REGION Network 2: MOVIMIENTO DE DATOS
   RUNG wire#powerrail
      Move(in := "FLUJO_FB_DB".SEÑAL_INGENIERIA, out1 => "flujo")
   END_RUNG
   RUNG wire#powerrail
      Move(in := "PRESION_LIQUIDO_FB_DB".SEÑAL_INGENIERIA, out1 => "presion")
   END_RUNG
   RUNG wire#powerrail
      Move(in := "valvula", out1 => "Consigna apertura Valvula Proporcional")
   END_RUNG
   RUNG wire#powerrail
      Move(in := "TEMPERATURA_FB_DB".SEÑAL_INGENIERIA, out1 => "temperatura")
   END_RUNG
   RUNG wire#powerrail
      Move(in := "PESO_FB_DB".SEÑAL_INGENIERIA, out1 => "peso tanque")
   END_RUNG
   RUNG wire#powerrail
      Move(in := "NIVEL_FB_DB".SEÑAL_INGENIERIA, out1 => "nivel_tanque")
   END_RUNG
   RUNG wire#powerrail
      Move(in := "bomba", out1 => "Consigna Velocidad Variador")
   END_RUNG
   // the same network as SCL:
   "flujo" := "FLUJO_FB_DB".SEÑAL_INGENIERIA;
   "presion" := "PRESION_LIQUIDO_FB_DB".SEÑAL_INGENIERIA;
   "Consigna apertura Valvula Proporcional" := "valvula";
   "temperatura" := "TEMPERATURA_FB_DB".SEÑAL_INGENIERIA;
   "peso tanque" := "PESO_FB_DB".SEÑAL_INGENIERIA;
   "nivel_tanque" := "NIVEL_FB_DB".SEÑAL_INGENIERIA;
   "Consigna Velocidad Variador" := "bomba";
END_REGION

REGION Network 3: PID NIVEL
   RUNG wire#powerrail
      Contact( "Tag_12" )
      "Smith_please_DB_1"(Sensor := "nivel_cal", Ref := "ref_lgr_nivel", Bomba => "bomba")
   END_RUNG
   // the same network as SCL:
   IF "Tag_12" THEN
       "Smith_please_DB_1"(Sensor := "nivel_cal", Ref := "ref_lgr_nivel", Bomba => "bomba");   // "Smith_please"
   END_IF;
END_REGION

REGION Network 4: ALARMAS
   RUNG wire#powerrail
      "ALARMAS"()
   END_RUNG
   // the same network as SCL:
   "ALARMAS"();
END_REGION

REGION Network 5: CARACTERIZACION Y CALIBRACION
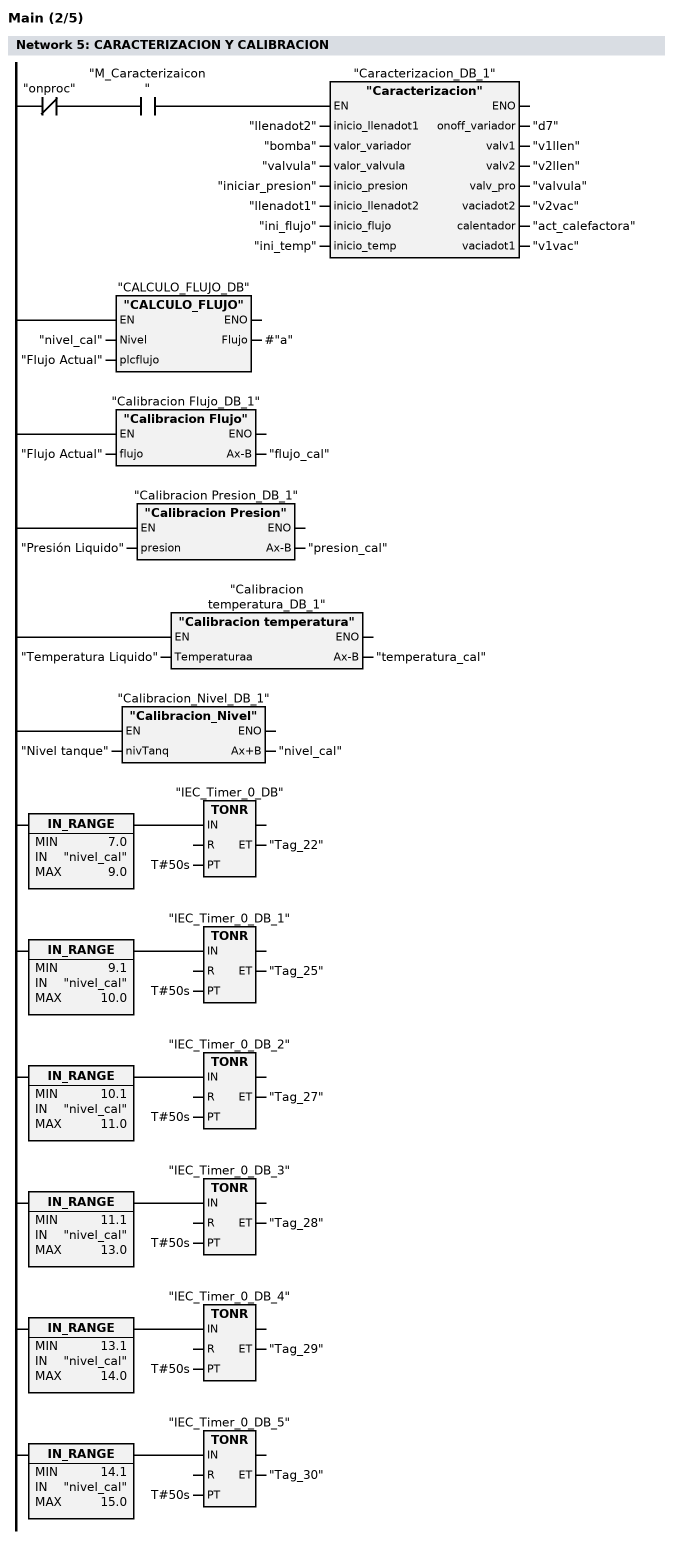
   IF NOT "onproc" AND "M_Caracterizaicon" THEN
       "Caracterizacion_DB_1"(inicio_llenadot1 := "llenadot2",   // "Caracterizacion"
                              valor_variador := "bomba",
                              valor_valvula := "valvula",
                              inicio_presion := "iniciar_presion",
                              inicio_llenadot2 := "llenadot1",
                              inicio_flujo := "ini_flujo",
                              inicio_temp := "ini_temp",
                              onoff_variador => "d7",
                              valv1 => "v1llen",
                              valv2 => "v2llen",
                              valv_pro => "valvula",
                              vaciadot2 => "v2vac",
                              calentador => "act_calefactora",
                              vaciadot1 => "v1vac");
   END_IF;
   "CALCULO_FLUJO_DB"(Nivel := "nivel_cal", plcflujo := "Flujo Actual", Flujo => #"a");   // "CALCULO_FLUJO"
   "Calibracion Flujo_DB_1"(flujo := "Flujo Actual", "Ax-B" => "flujo_cal");   // "Calibracion Flujo"
   "Calibracion Presion_DB_1"(presion := "Presión Liquido", "Ax-B" => "presion_cal");   // "Calibracion Presion"
   "Calibracion temperatura_DB_1"(Temperaturaa := "Temperatura Liquido", "Ax-B" => "temperatura_cal");   // "Calibracion temperatura"
   "Calibracion_Nivel_DB_1"(nivTanq := "Nivel tanque", "Ax+B" => "nivel_cal");   // "Calibracion_Nivel"
   "IEC_Timer_0_DB".TONR(IN := (7.0 <= "nivel_cal") AND ("nivel_cal" <= 9.0), PT := T#50s, ET => "Tag_22");
   "IEC_Timer_0_DB_1".TONR(IN := (9.1 <= "nivel_cal") AND ("nivel_cal" <= 10.0), PT := T#50s, ET => "Tag_25");
   "IEC_Timer_0_DB_2".TONR(IN := (10.1 <= "nivel_cal") AND ("nivel_cal" <= 11.0), PT := T#50s, ET => "Tag_27");
   "IEC_Timer_0_DB_3".TONR(IN := (11.1 <= "nivel_cal") AND ("nivel_cal" <= 13.0), PT := T#50s, ET => "Tag_28");
   "IEC_Timer_0_DB_4".TONR(IN := (13.1 <= "nivel_cal") AND ("nivel_cal" <= 14.0), PT := T#50s, ET => "Tag_29");
   "IEC_Timer_0_DB_5".TONR(IN := (14.1 <= "nivel_cal") AND ("nivel_cal" <= 15.0), PT := T#50s, ET => "Tag_30");
END_REGION

REGION Network 6: ON OFF PESO
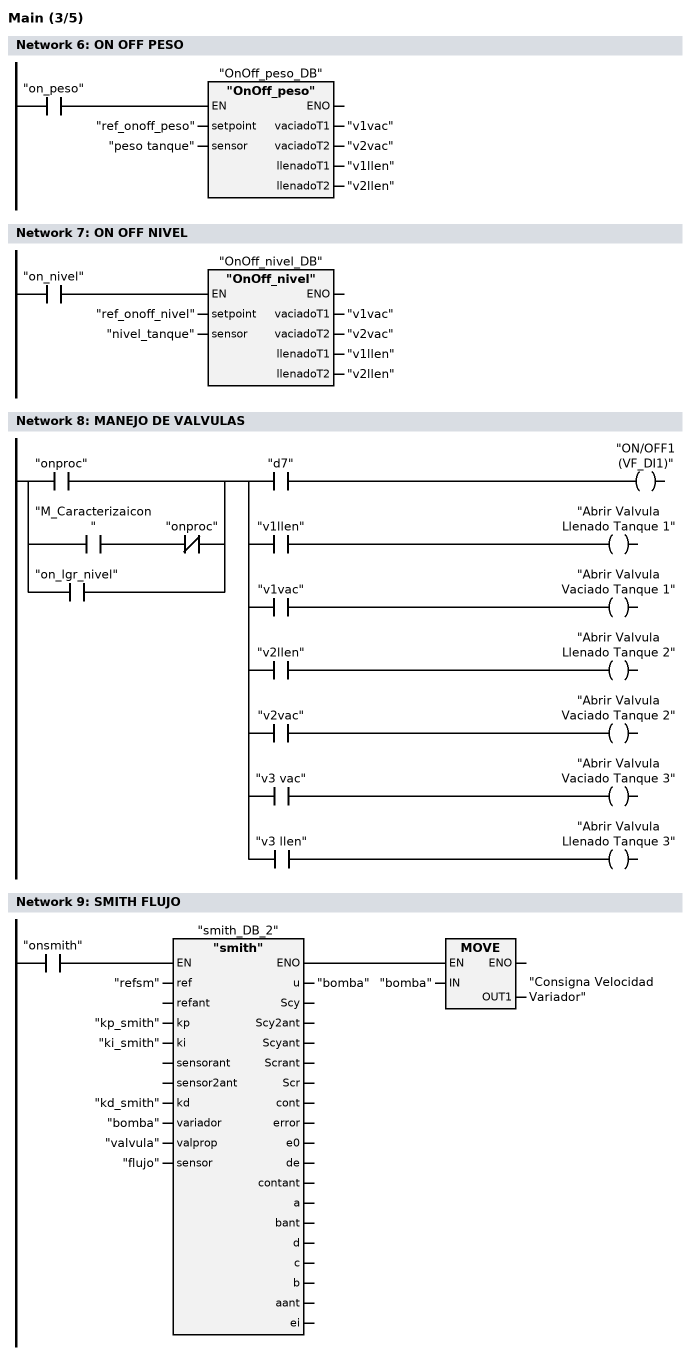
   RUNG wire#powerrail
      Contact( "on_peso" )
      "OnOff_peso_DB"(setpoint := "ref_onoff_peso", sensor := "peso tanque", vaciadoT1 => "v1vac", vaciadoT2 => "v2vac", llenadoT1 => "v1llen", llenadoT2 => "v2llen")
   END_RUNG
   // the same network as SCL:
   IF "on_peso" THEN
       "OnOff_peso_DB"(setpoint := "ref_onoff_peso",   // "OnOff_peso"
                       sensor := "peso tanque",
                       vaciadoT1 => "v1vac",
                       vaciadoT2 => "v2vac",
                       llenadoT1 => "v1llen",
                       llenadoT2 => "v2llen");
   END_IF;
END_REGION

REGION Network 7: ON OFF NIVEL
   RUNG wire#powerrail
      Contact( "on_nivel" )
      "OnOff_nivel_DB"(setpoint := "ref_onoff_nivel", sensor := "nivel_tanque", vaciadoT1 => "v1vac", vaciadoT2 => "v2vac", llenadoT1 => "v1llen", llenadoT2 => "v2llen")
   END_RUNG
   // the same network as SCL:
   IF "on_nivel" THEN
       "OnOff_nivel_DB"(setpoint := "ref_onoff_nivel",   // "OnOff_nivel"
                        sensor := "nivel_tanque",
                        vaciadoT1 => "v1vac",
                        vaciadoT2 => "v2vac",
                        llenadoT1 => "v1llen",
                        llenadoT2 => "v2llen");
   END_IF;
END_REGION

REGION Network 8: MANEJO DE VALVULAS
   RUNG wire#powerrail
      Contact( "onproc" )
      wire#w1
      Contact( "d7" )
      Coil( "ON/OFF1 (VF_DI1)" )
   END_RUNG
   RUNG wire#powerrail
      Contact( "M_Caracterizaicon" )
      I_Contact( "onproc" )
   END_RUNG wire#w1
   RUNG wire#powerrail
      Contact( "on_lgr_nivel" )
   END_RUNG wire#w1
   RUNG wire#w1
      Contact( "v1llen" )
      Coil( "Abrir Valvula Llenado Tanque 1" )
   END_RUNG
   RUNG wire#w1
      Contact( "v1vac" )
      Coil( "Abrir Valvula Vaciado Tanque 1" )
   END_RUNG
   RUNG wire#w1
      Contact( "v2llen" )
      Coil( "Abrir Valvula Llenado Tanque 2" )
   END_RUNG
   RUNG wire#w1
      Contact( "v2vac" )
      Coil( "Abrir Valvula Vaciado Tanque 2" )
   END_RUNG
   RUNG wire#w1
      Contact( "v3 vac" )
      Coil( "Abrir Valvula Vaciado Tanque 3" )
   END_RUNG
   RUNG wire#w1
      Contact( "v3 llen" )
      Coil( "Abrir Valvula Llenado Tanque 3" )
   END_RUNG
   // the same network as SCL:
   #_w1 := "onproc" OR ("M_Caracterizaicon" AND NOT "onproc") OR "on_lgr_nivel";
   "ON/OFF1 (VF_DI1)" := #_w1 AND "d7";
   "Abrir Valvula Llenado Tanque 1" := #_w1 AND "v1llen";
   "Abrir Valvula Vaciado Tanque 1" := #_w1 AND "v1vac";
   "Abrir Valvula Llenado Tanque 2" := #_w1 AND "v2llen";
   "Abrir Valvula Vaciado Tanque 2" := #_w1 AND "v2vac";
   "Abrir Valvula Vaciado Tanque 3" := #_w1 AND "v3 vac";
   "Abrir Valvula Llenado Tanque 3" := #_w1 AND "v3 llen";
END_REGION

REGION Network 9: SMITH FLUJO
   RUNG wire#powerrail
      Contact( "onsmith" )
      "smith_DB_2"(ref := "refsm", refant :=, kp := "kp_smith", ki := "ki_smith", sensorant :=, sensor2ant :=, kd := "kd_smith", variador := "bomba", valprop := "valvula", sensor := "flujo", u => "bomba", Scy =>, Scy2ant =>, Scyant =>, Scrant =>, Scr =>, cont =>, error =>, e0 =>, de =>, contant =>, "a" =>, bant =>, d =>, c =>, "b" =>, aant =>, ei =>)
      Move(in := "bomba", out1 => "Consigna Velocidad Variador")
   END_RUNG
   // the same network as SCL:
   "smith_DB_2"(EN := "onsmith",   // "smith"
                ref := "refsm",
                kp := "kp_smith",
                ki := "ki_smith",
                kd := "kd_smith",
                variador := "bomba",
                valprop := "valvula",
                sensor := "flujo",
                u => "bomba",
                ENO => #_w1);
   IF #_w1 THEN "Consigna Velocidad Variador" := "bomba"; END_IF;
END_REGION

REGION Network 10: ON OFF TEMPERATURA
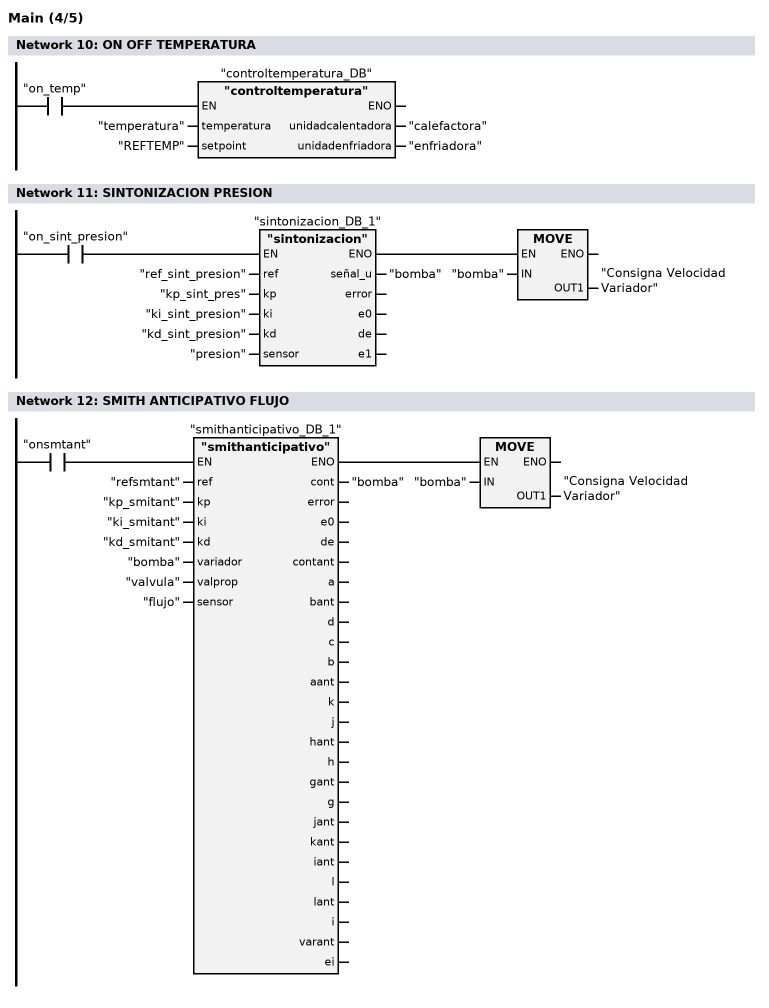
   RUNG wire#powerrail
      Contact( "on_temp" )
      "controltemperatura_DB"(temperatura := "temperatura", setpoint := "REFTEMP", unidadcalentadora => "calefactora", unidadenfriadora => "enfriadora")
   END_RUNG
   // the same network as SCL:
   IF "on_temp" THEN
       "controltemperatura_DB"(temperatura := "temperatura",   // "controltemperatura"
                               setpoint := "REFTEMP",
                               unidadcalentadora => "calefactora",
                               unidadenfriadora => "enfriadora");
   END_IF;
END_REGION

REGION Network 11: SINTONIZACION PRESION
   RUNG wire#powerrail
      Contact( "on_sint_presion" )
      "sintonizacion_DB_1"(ref := "ref_sint_presion", kp := "kp_sint_pres", ki := "ki_sint_presion", kd := "kd_sint_presion", sensor := "presion", señal_u => "bomba", error =>, e0 =>, de =>, e1 =>)
      Move(in := "bomba", out1 => "Consigna Velocidad Variador")
   END_RUNG
   // the same network as SCL:
   "sintonizacion_DB_1"(EN := "on_sint_presion",   // "sintonizacion"
                        ref := "ref_sint_presion",
                        kp := "kp_sint_pres",
                        ki := "ki_sint_presion",
                        kd := "kd_sint_presion",
                        sensor := "presion",
                        señal_u => "bomba",
                        ENO => #_w1);
   IF #_w1 THEN "Consigna Velocidad Variador" := "bomba"; END_IF;
END_REGION

REGION Network 12: SMITH ANTICIPATIVO FLUJO
   RUNG wire#powerrail
      Contact( "onsmtant" )
      "smithanticipativo_DB_1"(ref := "refsmtant", kp := "kp_smitant", ki := "ki_smitant", kd := "kd_smitant", variador := "bomba", valprop := "valvula", sensor := "flujo", cont => "bomba", error =>, e0 =>, de =>, contant =>, "a" =>, bant =>, d =>, c =>, "b" =>, aant =>, k =>, j =>, hant =>, h =>, gant =>, g =>, jant =>, kant =>, iant =>, l =>, lant =>, i =>, varant =>, ei =>)
      Move(in := "bomba", out1 => "Consigna Velocidad Variador")
   END_RUNG
   // the same network as SCL:
   "smithanticipativo_DB_1"(EN := "onsmtant",   // "smithanticipativo"
                           ref := "refsmtant",
                           kp := "kp_smitant",
                           ki := "ki_smitant",
                           kd := "kd_smitant",
                           variador := "bomba",
                           valprop := "valvula",
                           sensor := "flujo",
                           cont => "bomba",
                           ENO => #_w1);
   IF #_w1 THEN "Consigna Velocidad Variador" := "bomba"; END_IF;
END_REGION

REGION Network 13: FUZZY PRESION
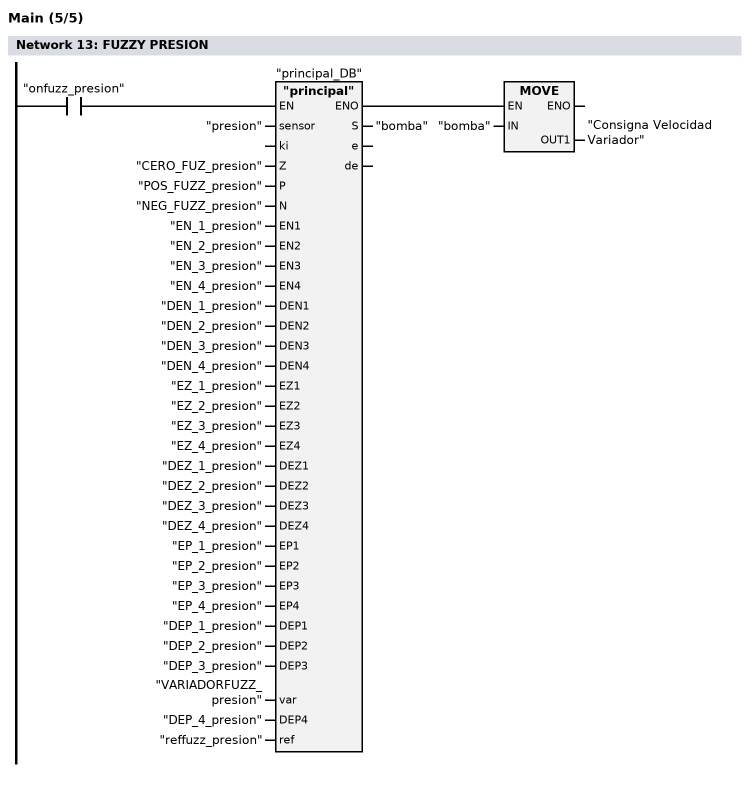
   RUNG wire#powerrail
      Contact( "onfuzz_presion" )
      "principal_DB"(sensor := "presion", ki :=, Z := "CERO_FUZ_presion", P := "POS_FUZZ_presion", N := "NEG_FUZZ_presion", EN1 := "EN_1_presion", EN2 := "EN_2_presion", EN3 := "EN_3_presion", EN4 := "EN_4_presion", DEN1 := "DEN_1_presion", DEN2 := "DEN_2_presion", DEN3 := "DEN_3_presion", DEN4 := "DEN_4_presion", EZ1 := "EZ_1_presion", EZ2 := "EZ_2_presion", EZ3 := "EZ_3_presion", EZ4 := "EZ_4_presion", DEZ1 := "DEZ_1_presion", DEZ2 := "DEZ_2_presion", DEZ3 := "DEZ_3_presion", DEZ4 := "DEZ_4_presion", EP1 := "EP_1_presion", EP2 := "EP_2_presion", EP3 := "EP_3_presion", EP4 := "EP_4_presion", DEP1 := "DEP_1_presion", DEP2 := "DEP_2_presion", DEP3 := "DEP_3_presion", var := "VARIADORFUZZ_presion", DEP4 := "DEP_4_presion", ref := "reffuzz_presion", S => "bomba", "e" =>, de =>)
      Move(in := "bomba", out1 => "Consigna Velocidad Variador")
   END_RUNG
   // the same network as SCL:
   "principal_DB"(EN := "onfuzz_presion",   // "principal"
                  sensor := "presion",
                  Z := "CERO_FUZ_presion",
                  P := "POS_FUZZ_presion",
                  N := "NEG_FUZZ_presion",
                  EN1 := "EN_1_presion",
                  EN2 := "EN_2_presion",
                  EN3 := "EN_3_presion",
                  EN4 := "EN_4_presion",
                  DEN1 := "DEN_1_presion",
                  DEN2 := "DEN_2_presion",
                  DEN3 := "DEN_3_presion",
                  DEN4 := "DEN_4_presion",
                  EZ1 := "EZ_1_presion",
                  EZ2 := "EZ_2_presion",
                  EZ3 := "EZ_3_presion",
                  EZ4 := "EZ_4_presion",
                  DEZ1 := "DEZ_1_presion",
                  DEZ2 := "DEZ_2_presion",
                  DEZ3 := "DEZ_3_presion",
                  DEZ4 := "DEZ_4_presion",
                  EP1 := "EP_1_presion",
                  EP2 := "EP_2_presion",
                  EP3 := "EP_3_presion",
                  EP4 := "EP_4_presion",
                  DEP1 := "DEP_1_presion",
                  DEP2 := "DEP_2_presion",
                  DEP3 := "DEP_3_presion",
                  var := "VARIADORFUZZ_presion",
                  DEP4 := "DEP_4_presion",
                  ref := "reffuzz_presion",
                  S => "bomba",
                  ENO => #_w1);
   IF #_w1 THEN "Consigna Velocidad Variador" := "bomba"; END_IF;
END_REGION
END_ORGANIZATION_BLOCK

ORGANIZATION_BLOCK "Cyclic interrupt"   // OB30, LAD, CyclicInterrupt
{ S7_Optimized_Access := 'TRUE' }
VERSION : 0.1
   VAR_INPUT
      Initial_Call : Bool;   // Initial call of this OB
      Event_Count : Int;   // Events discarded
   END_VAR
   VAR_TEMP
      PIDDT : Bool;
   END_VAR
BEGIN

REGION Network 2
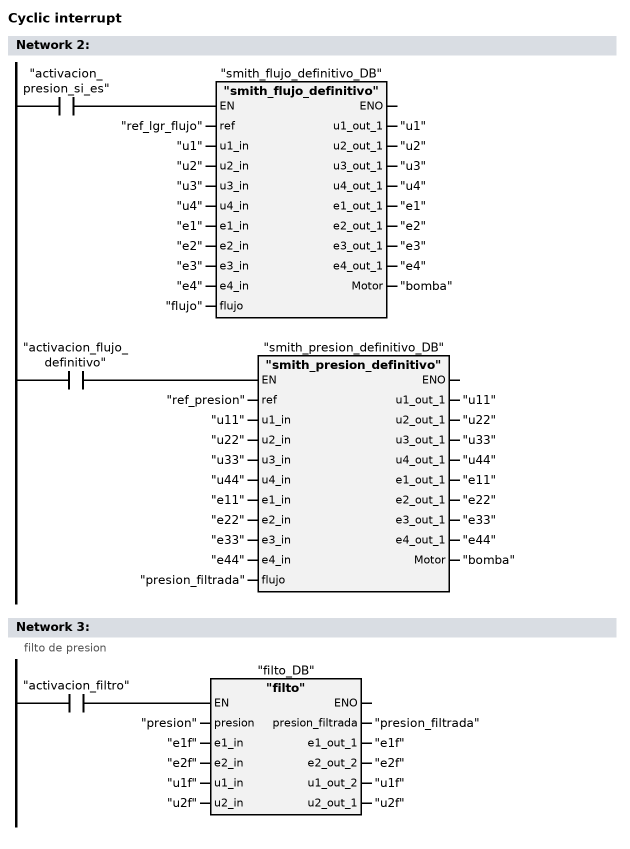
   RUNG wire#powerrail
      Contact( "activacion_presion_si_es" )
      "smith_flujo_definitivo_DB"(ref := "ref_lgr_flujo", u1_in := "u1", u2_in := "u2", u3_in := "u3", u4_in := "u4", e1_in := "e1", e2_in := "e2", e3_in := "e3", e4_in := "e4", flujo := "flujo", u1_out_1 => "u1", u2_out_1 => "u2", u3_out_1 => "u3", u4_out_1 => "u4", e1_out_1 => "e1", e2_out_1 => "e2", e3_out_1 => "e3", e4_out_1 => "e4", Motor => "bomba")
   END_RUNG
   RUNG wire#powerrail
      Contact( "activacion_flujo_definitivo" )
      "smith_presion_definitivo_DB"(ref := "ref_presion", u1_in := "u11", u2_in := "u22", u3_in := "u33", u4_in := "u44", e1_in := "e11", e2_in := "e22", e3_in := "e33", e4_in := "e44", flujo := "presion_filtrada", u1_out_1 => "u11", u2_out_1 => "u22", u3_out_1 => "u33", u4_out_1 => "u44", e1_out_1 => "e11", e2_out_1 => "e22", e3_out_1 => "e33", e4_out_1 => "e44", Motor => "bomba")
   END_RUNG
   // the same network as SCL:
   IF "activacion_presion_si_es" THEN
       "smith_flujo_definitivo_DB"(ref := "ref_lgr_flujo",   // "smith_flujo_definitivo"
                               u1_in := "u1",
                               u2_in := "u2",
                               u3_in := "u3",
                               u4_in := "u4",
                               e1_in := "e1",
                               e2_in := "e2",
                               e3_in := "e3",
                               e4_in := "e4",
                               flujo := "flujo",
                               u1_out_1 => "u1",
                               u2_out_1 => "u2",
                               u3_out_1 => "u3",
                               u4_out_1 => "u4",
                               e1_out_1 => "e1",
                               e2_out_1 => "e2",
                               e3_out_1 => "e3",
                               e4_out_1 => "e4",
                               Motor => "bomba");
   END_IF;
   IF "activacion_flujo_definitivo" THEN
       "smith_presion_definitivo_DB"(ref := "ref_presion",   // "smith_presion_definitivo"
                               u1_in := "u11",
                               u2_in := "u22",
                               u3_in := "u33",
                               u4_in := "u44",
                               e1_in := "e11",
                               e2_in := "e22",
                               e3_in := "e33",
                               e4_in := "e44",
                               flujo := "presion_filtrada",
                               u1_out_1 => "u11",
                               u2_out_1 => "u22",
                               u3_out_1 => "u33",
                               u4_out_1 => "u44",
                               e1_out_1 => "e11",
                               e2_out_1 => "e22",
                               e3_out_1 => "e33",
                               e4_out_1 => "e44",
                               Motor => "bomba");
   END_IF;
END_REGION

REGION Network 3
   // filto de presion
   RUNG wire#powerrail
      Contact( "activacion_filtro" )
      "filto_DB"(presion := "presion", e1_in := "e1f", e2_in := "e2f", u1_in := "u1f", u2_in := "u2f", presion_filtrada => "presion_filtrada", e1_out_1 => "e1f", e2_out_2 => "e2f", u1_out_2 => "u1f", u2_out_1 => "u2f")
   END_RUNG
   // the same network as SCL:
   IF "activacion_filtro" THEN
       "filto_DB"(presion := "presion",   // "filto"
                  e1_in := "e1f",
                  e2_in := "e2f",
                  u1_in := "u1f",
                  u2_in := "u2f",
                  presion_filtrada => "presion_filtrada",
                  e1_out_1 => "e1f",
                  e2_out_2 => "e2f",
                  u1_out_2 => "u1f",
                  u2_out_1 => "u2f");
   END_IF;
END_REGION
END_ORGANIZATION_BLOCK

ORGANIZATION_BLOCK "Startup"   // OB100, LAD, Startup
TITLE = "Complete Restart"
{ S7_Optimized_Access := 'TRUE' }
VERSION : 0.1
   VAR_INPUT
      LostRetentive : Bool;   // True if retentive data are lost
      LostRTC : Bool;   // True if date and time are lost
   END_VAR
BEGIN

REGION Network 1
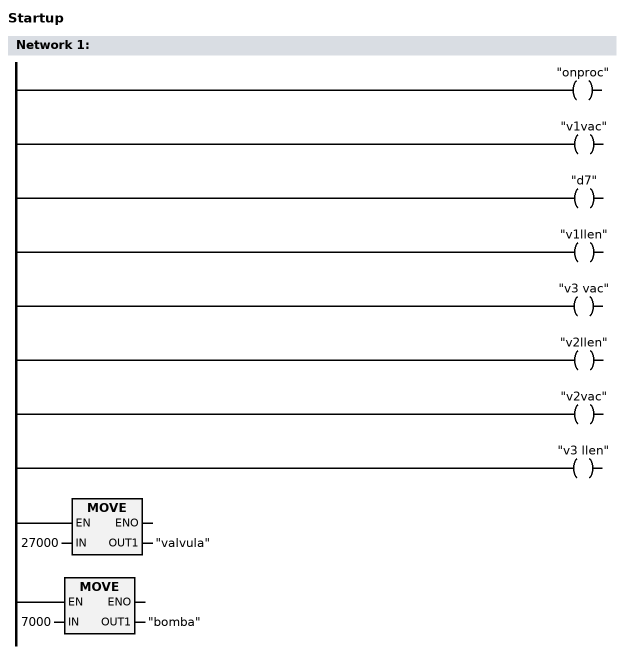
   RUNG wire#powerrail
      Coil( "onproc" )
   END_RUNG
   RUNG wire#powerrail
      Coil( "v1vac" )
   END_RUNG
   RUNG wire#powerrail
      Coil( "d7" )
   END_RUNG
   RUNG wire#powerrail
      Coil( "v1llen" )
   END_RUNG
   RUNG wire#powerrail
      Coil( "v3 vac" )
   END_RUNG
   RUNG wire#powerrail
      Coil( "v2llen" )
   END_RUNG
   RUNG wire#powerrail
      Coil( "v2vac" )
   END_RUNG
   RUNG wire#powerrail
      Coil( "v3 llen" )
   END_RUNG
   RUNG wire#powerrail
      Move(in := 27000, out1 => "valvula")
   END_RUNG
   RUNG wire#powerrail
      Move(in := 7000, out1 => "bomba")
   END_RUNG
   // the same network as SCL:
   "onproc" := TRUE;
   "v1vac" := TRUE;
   "d7" := TRUE;
   "v1llen" := TRUE;
   "v3 vac" := TRUE;
   "v2llen" := TRUE;
   "v2vac" := TRUE;
   "v3 llen" := TRUE;
   "valvula" := 27000;
   "bomba" := 7000;
END_REGION
END_ORGANIZATION_BLOCK

(* ===== HMI "HMI_RT_1" =====
system functions are stored by id; their names below are inferred from use
connection "HMI_Conexión_2": ETHERNET, S7_1500_OMS

HMI tags "Tabla de variables estándar"
   "Número_imagen_variable" : UInt, internal
   "v1llen" : Bool = PLC v1llen AT %M2.3, 1 s
   "v1vac" : Bool = PLC v1vac AT %M2.4, 1 s
   "v2llen" : Bool = PLC v2llen AT %M2.5, 1 s
   "v2vac" : Bool = PLC v2vac AT %M2.6, 1 s
   "v3" : Bool = PLC "v3 vac" AT %M5.0, 1 s
   "valvula" : Int = PLC valvula AT %MW8, 1 s
   "onproc" : Bool = PLC onproc AT %M2.7, 1 s
   "d7" : Bool = PLC d7 AT %M3.0, 1 s
   "bomba" : Int = PLC bomba AT %MW6, 1 s
   "onsint" : Bool = PLC onsint AT %M5.3, 1 s
   "onfuzz" : Bool = PLC onfuzz AT %M5.1, 1 s
   "Nivel tanque" : Int = PLC "Nivel tanque" AT %IW112, 1 s
   "velmotor" : Word = PLC velmotor AT %MW26, 1 s
   "presion" : Real = PLC presion AT %MD10, 1 s
   "flujo" : Real = PLC flujo AT %MD14, 1 s
   "refsint" : Real = PLC refsint AT %MD24, 1 s
   "reflgr" : Real = PLC reflgr AT %MD26, 1 s
   "onlgr" : Bool = PLC onlgr AT %M5.6, 1 s
   "onsmith" : Bool = PLC onsmith AT %M5.4, 1 s
   "onsmtant" : Bool = PLC onsmtant AT %M5.5, 1 s
   "refsmtant" : Real = PLC refsmtant AT %MD28, 1 s
   "reffuzz" : Real = PLC reffuzz AT %MD22, 1 s
   "temperatura" : Real = PLC temperatura AT %MD16, 1 s
   "REFTEMP" : Real = PLC REFTEMP AT %MD30, 1 s
   "on_temp" : Bool = PLC on_temp AT %M5.7, 1 s
   "Activar Unidad Enfriadora" : Bool = PLC "Activar Unidad Enfriadora" AT %Q1.7, 1 s
   "Activar Unidad Calefactora" : Bool = PLC "Activar Unidad Calefactora" AT %Q1.6, 1 s
   "Abrir Valvula Vaciado Tanque 3" : Bool = PLC "Abrir Valvula Vaciado Tanque 3" AT %Q1.5, 1 s
   "Abrir Valvula Llenado Tanque 3" : Bool = PLC "Abrir Valvula Llenado Tanque 3" AT %Q1.4, 1 s
   "Temperatura Liquido" : Int = PLC "Temperatura Liquido" AT %IW106, 1 s
   "kp_sint" : Real = PLC kp_sint AT %MD34, 1 s
   "ki_sint" : Real = PLC ki_sint AT %MD38, 1 s
   "kd_sint" : Real = PLC kd_sint AT %MD42, 1 s
   "Consigna apertura Valvula Proporcional" : Int = PLC "Consigna apertura Valvula Proporcional" AT %QW106, 1 s
   "Consigna Velocidad Variador" : Int = PLC "Consigna Velocidad Variador" AT %QW104, 1 s
   "Switch de Nivel Alto Tanque 1 (NC)" : Bool = PLC "Switch de Nivel Alto Tanque 1 (NC)" AT %I1.3, 1 s
   "Switch de Nivel Bajo Tanque 1 (NO)" : Bool = PLC "Switch de Nivel Bajo Tanque 1 (NO)" AT %I1.2, 1 s
   "Abrir Valvula Llenado Tanque 1" : Bool = PLC "Abrir Valvula Llenado Tanque 1" AT %Q1.0, 1 s
   "Abrir Valvula Llenado Tanque 2" : Bool = PLC "Abrir Valvula Llenado Tanque 2" AT %Q1.2, 1 s
   "Abrir Valvula Vaciado Tanque 1" : Bool = PLC "Abrir Valvula Vaciado Tanque 1" AT %Q1.1, 1 s
   "Abrir Valvula Vaciado Tanque 2" : Bool = PLC "Abrir Valvula Vaciado Tanque 2" AT %Q1.3, 1 s
   "kp_lgr" : Real = PLC kp_lgr AT %MD46, 1 s
   "ki_lgr" : Real = PLC ki_lgr AT %MD54, 1 s
   "kd_lgr" : Real = PLC kd_lgr AT %MD58, 1 s
   "refsm" : Real = PLC refsm AT %MD20, 1 s
   "kp_smith" : Real = PLC kp_smith AT %MD62, 1 s
   "ki_smith" : Real = PLC ki_smith AT %MD66, 1 s
   "kd_smith" : Real = PLC kd_smith AT %MD70, 1 s
   "kp_smitant" : Real = PLC kp_smitant AT %MD74, 1 s
   "ki_smitant" : Real = PLC ki_smitant AT %MD78, 1 s
   "kd_smitant" : Real = PLC kd_smitant AT %MD82, 1 s
   "EN_1" : Real = PLC EN_1 AT %MD98, 1 s
   "EN_2" : Real = PLC EN_2 AT %MD102, 1 s
   "EN_3" : Real = PLC EN_3 AT %MD106, 1 s
   "EN_4" : Real = PLC EN_4 AT %MD110, 1 s
   "EZ_1" : Real = PLC EZ_1 AT %MD130, 1 s
   "EZ_2" : Real = PLC EZ_2 AT %MD134, 1 s
   "EZ_3" : Real = PLC EZ_3 AT %MD138, 1 s
   "EZ_4" : Real = PLC EZ_4 AT %MD142, 1 s
   "EP_1" : Real = PLC EP_1 AT %MD162, 1 s
   "EP_2" : Real = PLC EP_2 AT %MD166, 1 s
   "EP_3" : Real = PLC EP_3 AT %MD170, 1 s
   "EP_4" : Real = PLC EP_4 AT %MD174, 1 s
   "DEN_1" : Real = PLC DEN_1 AT %MD114, 1 s
   "DEN_2" : Real = PLC DEN_2 AT %MD118, 1 s
   "DEN_3" : Real = PLC DEN_3 AT %MD122, 1 s
   "DEN_4" : Real = PLC DEN_4 AT %MD126, 1 s
   "DEZ_1" : Real = PLC DEZ_1 AT %MD146, 1 s
   "DEZ_2" : Real = PLC DEZ_2 AT %MD150, 1 s
   "DEZ_3" : Real = PLC DEZ_3 AT %MD154, 1 s
   "DEZ_4" : Real = PLC DEZ_4 AT %MD158, 1 s
   "DEP_1" : Real = PLC DEP_1 AT %MD178, 1 s
   "DEP_2" : Real = PLC DEP_2 AT %MD182, 1 s
   "DEP_3" : Real = PLC DEP_3 AT %MD186, 1 s
   "DEP_4" : Real = PLC DEP_4 AT %MD194, 1 s
   "NEG_FUZZ" : Real = PLC NEG_FUZZ AT %MD94, 1 s
   "CERO_FUZ" : Real = PLC CERO_FUZ AT %MD86, 1 s
   "POS_FUZZ" : Real = PLC POS_FUZZ AT %MD90, 1 s
   "VARIADORFUZZ" : Real = PLC VARIADORFUZZ AT %MD190, 1 s
   "v3 llen" : Bool = PLC "v3 llen" AT %M8.0, 1 s
   "enfriadora" : Bool = PLC enfriadora AT %M7.0, 1 s
   "calefactora" : Bool = PLC calefactora AT %M6.0, 1 s
   "on_lgr_flujo" : Bool = PLC on_lgr_flujo AT %M2.1, 1 s
   "ref_lgr_flujo" : Real = PLC ref_lgr_flujo AT %MD214, 1 s
   "kp_lgr_flujo" : Real = PLC kp_lgr_flujo AT %MD218, 1 s
   "ki_lgr_flujo" : Real = PLC ki_lgr_flujo AT %MD222, 1 s
   "kd_lgr_flujo" : Real = PLC kd_lgr_flujo AT %MD226, 1 s
   "on_sint_presion" : Bool = PLC on_sint_presion AT %M2.0, 1 s
   "ref_sint_presion" : Real = PLC ref_sint_presion AT %MD198, 1 s
   "kp_sint_pres" : Real = PLC kp_sint_pres AT %MD202, 1 s
   "ki_sint_presion" : Real = PLC ki_sint_presion AT %MD206, 1 s
   "kd_sint_presion" : Real = PLC kd_sint_presion AT %MD210, 1 s
   "onfuzz_presion" : Bool = PLC onfuzz_presion AT %M2.2, 1 s
   "reffuzz_presion" : Real = PLC reffuzz_presion AT %MD342, 1 s
   "NEG_FUZZ_presion" : Real = PLC NEG_FUZZ_presion AT %MD238, 1 s
   "CERO_FUZ_presion" : Real = PLC CERO_FUZ_presion AT %MD230, 1 s
   "POS_FUZZ_presion" : Real = PLC POS_FUZZ_presion AT %MD234, 1 s
   "VARIADORFUZZ_presion" : Real = PLC VARIADORFUZZ_presion AT %MD334, 1 s
   "EN_1_presion" : Real = PLC EN_1_presion AT %MD242, 1 s
   "EN_2_presion" : Real = PLC EN_2_presion AT %MD246, 1 s
   "EN_3_presion" : Real = PLC EN_3_presion AT %MD250, 1 s
   "EN_4_presion" : Real = PLC EN_4_presion AT %MD254, 1 s
   "EZ_1_presion" : Real = PLC EZ_1_presion AT %MD274, 1 s
   "EZ_2_presion" : Real = PLC EZ_2_presion AT %MD278, 1 s
   "EZ_3_presion" : Real = PLC EZ_3_presion AT %MD282, 1 s
   "EZ_4_presion" : Real = PLC EZ_4_presion AT %MD286, 1 s
   "EP_1_presion" : Real = PLC EP_1_presion AT %MD306, 1 s
   "EP_2_presion" : Real = PLC EP_2_presion AT %MD310, 1 s
   "EP_3_presion" : Real = PLC EP_3_presion AT %MD314, 1 s
   "EP_4_presion" : Real = PLC EP_4_presion AT %MD318, 1 s
   "DEN_1_presion" : Real = PLC DEN_1_presion AT %MD258, 1 s
   "DEN_2_presion" : Real = PLC DEN_2_presion AT %MD262, 1 s
   "DEN_3_presion" : Real = PLC DEN_3_presion AT %MD266, 1 s
   "DEN_4_presion" : Real = PLC DEN_4_presion AT %MD270, 1 s
   "DEZ_1_presion" : Real = PLC DEZ_1_presion AT %MD290, 1 s
   "DEZ_2_presion" : Real = PLC DEZ_2_presion AT %MD294, 1 s
   "DEZ_3_presion" : Real = PLC DEZ_3_presion AT %MD298, 1 s
   "DEZ_4_presion" : Real = PLC DEZ_4_presion AT %MD302, 1 s
   "DEP_1_presion" : Real = PLC DEP_1_presion AT %MD322, 1 s
   "DEP_2_presion" : Real = PLC DEP_2_presion AT %MD326, 1 s
   "DEP_3_presion" : Real = PLC DEP_3_presion AT %MD330, 1 s
   "DEP_4_presion" : Real = PLC DEP_4_presion AT %MD338, 1 s
   "ALARMA1" : Bool = PLC ALARMA1 AT %M200.0, 1 s
   "ALARMA_ALARMA1" : Int = PLC ALARMA.ALARMA1, 1 s
   "ref_onoff_peso" : Real = PLC ref_onoff_peso AT %MD374, 1 s
   "peso tanque" : Real = PLC "peso tanque" AT %MD370, 1 s
   "on_peso" : Bool = PLC on_peso AT %M3.5, 1 s
   "ref_onoff_nivel" : Real = PLC ref_onoff_nivel AT %MD366, 1 s
   "nivel_tanque" : Real = PLC nivel_tanque AT %MD346, 1 s
   "on_nivel" : Bool = PLC on_nivel AT %M3.4, 1 s
   "on_lgr_nivel" : Bool = PLC on_lgr_nivel AT %M3.3, 1 s
   "ref_lgr_nivel" : Real = PLC ref_lgr_nivel AT %MD350, 1 s
   "kp_lgr_nivel" : Real = PLC kp_lgr_nivel AT %MD354, 1 s
   "ki_lgr_nivel" : Real = PLC ki_lgr_nivel AT %MD358, 1 s
   "kd_lgr_nivel" : Real = PLC kd_lgr_nivel AT %MD362, 1 s
   "ALARMA_ALARMA2" : Int = PLC ALARMA.ALARMA2, 1 s
   "ALARMA_ALARMA3" : Int = PLC ALARMA.ALARMA3, 1 s
   "ALARMA_ALARMA4" : Int = PLC ALARMA.ALARMA4, 1 s
   "ALARMA_ALARMA5" : Int = PLC ALARMA.ALARMA5, 1 s
   "ALARMA_ALARMA6" : Int = PLC ALARMA.ALARMA6, 1 s
   "ALARMA_ALARMA7" : Int = PLC ALARMA.ALARMA7, 1 s
   "ALARMA_ALARMA8" : Int = PLC ALARMA.ALARMA8, 1 s
   "ALARMA_ALARMA9" : Int = PLC ALARMA.ALARMA9, 1 s
   "ALARMA_ALARMA10" : Int = PLC ALARMA.ALARMA10, 1 s
   "ALARMA_ALARMA11" : Int = PLC ALARMA.ALARMA11, 1 s
   "ALARMA_ALARMA12" : Int = PLC ALARMA.ALARMA12, 1 s
   "ALARMA_ALARMA13" : Int = PLC ALARMA.ALARMA13, 1 s
   "ALARMA_ALARMA14" : Int = PLC ALARMA.ALARMA14, 1 s
   "ALARMA_ALARMA15" : Int = PLC ALARMA.ALARMA15, 1 s
   "ALARMA_ALARMA16" : Int = PLC ALARMA.ALARMA16, 1 s
   "ALARMA_ALARMA17" : Int = PLC ALARMA.ALARMA17, 1 s
   "ALARMA_ALARMA18" : Int = PLC ALARMA.ALARMA18, 1 s
   "nivel_cal" : Real = PLC nivel_cal AT %MD394, 1 s

discrete alarms
   1: 'NIVEL DEL TANQUE 1 ALTO', class Errors, trigger "ALARMA_ALARMA1" bit 0
   2: 'NIVEL DEL TANQUE 1 BAJO', class Errors, trigger "ALARMA_ALARMA2" bit 1
   3: 'VALVULA PROPORCIONAL CERRADA', class Errors, trigger "ALARMA_ALARMA3" bit 0
   4: 'UN CONTROL EN FUNCIONAMIENTO', class Errors, trigger "ALARMA_ALARMA4" bit 0
   5: 'TEMPERATURA MUY ALTA', class Errors, trigger "ALARMA_ALARMA5" bit 0
   6: 'ENCENDER BOMBA', class Errors, trigger "ALARMA_ALARMA6" bit 0
   7: 'CONTROL ON-OFF TEMPERATURA ENCENDIDO', class Errors, trigger "ALARMA_ALARMA7" bit 0
   8: 'CONTROL ON-OFF PESO ENCENDIDO', class Errors, trigger "ALARMA_ALARMA8" bit 0
   9: 'CONTROL SINTONIZACION PRESION ENCENDIDO', class Errors, trigger "ALARMA_ALARMA9" bit 0
   10: 'CONTROL PID PRESION ENCENDIDO', class Errors, trigger "ALARMA_ALARMA10" bit 0
   11: 'CONTROL FUZZY PRESION ENCENDIDO', class Errors, trigger "ALARMA_ALARMA11" bit 0
   12: 'CONTROL SINTONIZACION FLUJO ENCENDIDO', class Errors, trigger "ALARMA_ALARMA12" bit 0
   13: 'CONTROL PID FLUJO ENCENDIDO', class Errors, trigger "ALARMA_ALARMA13" bit 0
   14: 'CONTROL SMITH FLUJO ENCENDIDO', class Errors, trigger "ALARMA_ALARMA14" bit 0
   15: 'CONTROL SMITH ANTICIPATIVO FLUJO ENCENDIDO', class Errors, trigger "ALARMA_ALARMA15" bit 0
   16: 'CONTROL FUZZY FLUJO ENCENDIDO', class Errors, trigger "ALARMA_ALARMA16" bit 0
   17: 'CONTROL ONOFF NIVEL ENCENDIDO', class Errors, trigger "ALARMA_ALARMA17" bit 0
   18: 'CONTROL PID NIVEL ENCENDIDO', class Errors, trigger "ALARMA_ALARMA18" bit 0

text list "Nombre_imagen_lista_texto": 1 'Imagen raíz'

screen "Imagen raíz" 1280x740, template "Plantilla_1"
   on GenerateScreen: SetTag("Número_imagen_variable", 1)
   TextField "HmiScreenItemData" at 0,8 size 1270x79; Text 'TÉCNICAS DE CONTROL Y SUPERVISION EN EL MODULO DE PROCESOS'
   TextField "HmiScreenItemData_1" at 0,56 size 1270x77; Text 'MODULO DE ENTRENAMIENTO #1'
   TextField "HmiScreenItemData_2" at 0,102 size 1270x71; Text '2018'
   TextField "HmiScreenItemData_3" at 0,281 size 1270x77; Text 'JOSE ANTONIO TUMIALAN BORJA'
   Button "Botón_1" at 452,587 size 372x68; TextOff 'INGRESO'
      on Click: ActivateScreen("Variables fisicas", 0)
   TextField "HmiScreenItemData_4" at 0,188 size 1270x77; Text 'MIGUEL ANGEL ROJAS MAHECHA'
   TextField "HmiScreenItemData_5" at 0,142 size 1270x77; Text 'ESTUDIANTE'
   TextField "HmiScreenItemData_6" at 0,234 size 1270x77; Text 'DIRECTOR'
   GraphicView "Visor de gráficos_2" at 479,357 size 299x153; Picture "LASALLEGI"

Template "Plantilla_1" 1280x740
   Button "Template_Button" at 1200,679 size 78x59; TextOff 'ExitRuntime'; PictureOff "ExitRuntime_TP1500_Comfort_TR"; PictureOn "ExitRuntime_TP1500_Comfort_TR"
      on Release: StopRuntime(0)
   Button "Template_Button_1" at 1120,679 size 78x59; TextOff 'Text'
   Button "Template_Button_2" at 1040,679 size 78x59; TextOff 'Text'
   Button "Template_Button_3" at 960,679 size 78x59; TextOff 'Text'
   Button "Template_Button_4" at 880,679 size 78x59; TextOff 'Text'
   Button "Template_Button_5" at 800,679 size 78x59; TextOff 'Text'
   Button "Template_Button_6" at 720,679 size 78x59; TextOff 'Text'
   Button "Template_Button_7" at 640,679 size 78x59; TextOff 'Text'
   Button "Template_Button_8" at 561,679 size 78x59; TextOff 'Text'
   Button "Template_Button_9" at 481,679 size 78x59; TextOff 'Text'
   Button "Template_Button_10" at 401,679 size 78x59; TextOff 'Text'
   Button "Template_Button_11" at 321,679 size 78x59; TextOff 'Text'
   Button "Template_Button_12" at 241,679 size 78x59; TextOff 'Text'
   Button "Template_Button_13" at 161,679 size 78x59; TextOff 'Text'
   Button "Template_Button_14" at 81,679 size 78x59; TextOff 'Text'
   Button "Template_Button_15" at 1,679 size 78x59; TextOff 'NavigateHome'; PictureOff "NavigateHome_TP1500_Comfort_TR"; PictureOn "NavigateHome_TP1500_Comfort_TR"
      on Release: ActivateScreen("Imagen raíz", 0)

screen "controles flujo" 1280x740
   TextField "Campo de texto_1" at 323,52 size 636x43; Text 'TECNICAS DE CONTROL PARA FLUJO'
   Button "Botón_1" at 111,168 size 304x122; TextOff 'SINTONIZACION'
      on Click: ActivateScreen("sintonizacion flujo", 0)
   Button "Botón_4" at 854,167 size 304x122; TextOff 'PREDICTOR SMITH'
      on Click: ActivateScreen("predictor smith flujo", 0)
   Button "Botón_5" at 112,345 size 304x122; TextOff 'SMITH-ANTICIPATIVO'
      on Click: ActivateScreen("smithant flujo", 0)
   Button "Botón_6" at 856,341 size 304x122; TextOff 'FUZZY'
      on Click: ActivateScreen("fuzzy flujo", 0)
   Button "Botón_7" at 488,576 size 304x104; TextOff 'REGRESAR'
      on Click: ActivateScreen("Variables fisicas", 0)
   Button "Botón_2" at 482,167 size 304x122; TextOff 'PID'
      on Click: ActivateScreen("lgr_flujo", 0)

screen "sintonizacion flujo" 1280x740
   Button "Botón_1" at 760,621 size 300x80; TextOff 'REGRESAR'
      on Click: ActivateScreen("controles flujo", 0)
   GraphicView "Visor de gráficos_7" at 499,243 size 138x216; Picture "Gráfico_11"
   GraphicView "Visor de gráficos_2" at 924,449 size 56x50; Picture "Gráfico_14"
   GraphicView "Visor de gráficos_3" at 554,448 size 53x52; Picture "Gráfico_15"
   GraphicView "Visor de gráficos_4" at 632,290 size 52x29; Picture "Gráfico_16"
   GraphicView "Visor de gráficos_9" at 381,509 size 123x85; Picture "Gráfico_19"
   GraphicView "Visor de gráficos_10" at 388,97 size 61x52; Picture "Gráfico_20"
   GraphicView "Visor de gráficos_11" at 525,67 size 33x57; Picture "Gráfico_21"
   GraphicView "Visor de gráficos_12" at 628,83 size 61x63; Picture "Gráfico_22"
   GraphicView "Visor de gráficos_15" at 681,256 size 62x64; Picture "Gráfico_23"
   GraphicView "Visor de gráficos_17" at 748,469 size 55x58; Picture "Gráfico_24"
   GraphicView "Visor de gráficos_18" at 739,263 size 53x56; Picture "Gráfico_25"
   GraphicView "Visor de gráficos_6" at 790,256 size 62x64; Picture "Gráfico_23"
   GraphicView "Visor de gráficos_19" at 850,290 size 52x29; Picture "Gráfico_16"
   GraphicView "Visor de gráficos_20" at 894,243 size 138x216; Picture "Gráfico_11"
   GraphicView "Visor de gráficos_21" at 603,471 size 92x29; Picture "Gráfico_16"
   GraphicView "Visor de gráficos_22" at 692,437 size 62x64; Picture "Gráfico_23"
   GraphicView "Visor de gráficos_24" at 801,437 size 62x64; Picture "Gráfico_23"
   GraphicView "Visor de gráficos_25" at 861,471 size 67x29; Picture "Gráfico_16"
   GraphicView "Visor de gráficos_1" at 734,515 size 56x50; Picture "Gráfico_14"
   GraphicView "Visor de gráficos_8" at 495,537 size 251x29; Picture "Gráfico_16"
   GraphicView "Visor de gráficos_13" at 306,490 size 54x52; Picture "Gráfico_15"
   GraphicView "Visor de gráficos_14" at 344,513 size 48x29; Picture "Gráfico_16"
   GraphicView "Visor de gráficos_16" at 353,115 size 38x29; Picture "Gráfico_16"
   GraphicView "Visor de gráficos_23" at 445,116 size 187x29; Picture "Gráfico_16"
   GraphicView "Visor de gráficos_26" at 435,221 size 46x68; Picture "Gráfico_26"
   GraphicView "Visor de gráficos_27" at 434,333 size 46x68; Picture "Gráfico_26"
   GraphicView "Visor de gráficos_28" at 462,279 size 45x10; Picture "Gráfico_16"
   GraphicView "Visor de gráficos_29" at 463,391 size 45x10; Picture "Gráfico_16"
   GraphicView "Visor de gráficos_30" at 304,155 size 31x344; Picture "Gráfico_17"
   GraphicView "Visor de gráficos_31" at 307,117 size 52x48; Picture "Gráfico_27"
   GraphicView "Visor de gráficos_32" at 683,116 size 60x29; Picture "Gráfico_16"
   GraphicView "Visor de gráficos_34" at 750,153 size 31x120; Picture "Gráfico_17"
   IOField "Campo ES_1" at 398,477 size 96x32; FormatPattern s99999
      ProcessValue <- "bomba"
   IOField "Campo ES_2" at 370,54 size 96x32; FormatPattern s999999999.999
      ProcessValue <- "flujo"
   IOField "Campo ES_3" at 611,36 size 96x32; FormatPattern s99999
      ProcessValue <- "valvula"
   IOField "Campo ES_4" at 495,149 size 96x32; FormatPattern s999999999.999
      ProcessValue <- "presion"
   Bar "Barra_1" at 900,275 size 131x145; MinimumValue 0; MaximumValue 27000
      ProcessValue <- "Nivel tanque"
   GraphicView "Visor de gráficos_35" at 930,200 size 75x76; Picture "Gráfico_28"
   TextField "Campo de texto_1" at 31,256 size 99x25; Text 'SETPOINT'
   TextField "Campo de texto_2" at 59,340 size 135x25; Text 'CONSTANTES'
   TextField "Campo de texto_3" at 55,406 size 43x25; Text 'KP:'
   TextField "Campo de texto_4" at 57,454 size 40x25; Text 'KI:'
   TextField "Campo de texto_5" at 57,502 size 39x25; Text 'KD:'
   Button "Botón_6" at 680,251 size 61x79; TextOff 'Text'
      on Click: InvertBit("v1llen")
   Button "Botón_7" at 692,431 size 61x79; TextOff 'Text'
      on Click: InvertBit("v1vac")
   Button "Botón_8" at 792,253 size 61x79; TextOff 'Text'
      on Click: InvertBit("v2llen")
   Button "Botón_9" at 800,431 size 65x83; TextOff 'Text'
      on Click: InvertBit("v2vac")
   TextField "Campo de texto_6" at 40,81 size 197x25; Text 'CONTROL DE FLUJO'
   TextField "Campo de texto_7" at 58,106 size 162x25; Text 'SINTONIZACION'
   IOField "Campo ES_6" at 137,251 size 100x40; FormatPattern s999999999.999
      ProcessValue <- "refsint"
   Button "Botón_2" at 40,173 size 108x49; TextOff 'ON'
      on Click: InvertBit("onsint"); ResetBit("on_temp"); ResetBit("onfuzz"); ResetBit("onlgr"); ResetBit("onsmith"); ResetBit("onsmtant")
   Circle "Círculo_5" at 181,180 size 36x36
      Appearance <- "onsint"
   Circle "Círculo_6" at 647,144 size 23x23
      Appearance <- "d7"
   Button "Botón_3" at 134,621 size 300x80; TextOff 'TENDENCIAS'
      on Click: ActivateScreen("tendencia sintonizacion flujo", 0)
   IOField "Campo ES_7" at 110,399 size 99x39; FormatPattern s999999999.999
      ProcessValue <- "kp_sint"
   IOField "Campo ES_8" at 108,452 size 99x39; FormatPattern s999999999.999
      ProcessValue <- "ki_sint"
   IOField "Campo ES_9" at 108,504 size 99x39; FormatPattern s999999999.999
      ProcessValue <- "kd_sint"
   GraphicView "Visor de gráficos_37" at 282,217 size 80x80; Picture "Gráfico_30"
   Circle "Círculo_7" at 374,241 size 23x23
      Appearance <- "Activar Unidad Enfriadora"
   Circle "Círculo_8" at 379,403 size 23x23
      Appearance <- "Activar Unidad Calefactora"
   Button "Botón_5" at 280,216 size 82x80; TextOff 'Text'
      on Click: InvertBit("enfriadora")
   GraphicView "Visor de gráficos_36" at 282,365 size 80x80; Picture "Gráfico_31"
   Button "Botón_10" at 282,362 size 83x87; TextOff 'Text'
      on Click: InvertBit("calefactora")
   Rectangle "Rectángulo_2" at 444,225 size 33x20
      Appearance <- "Switch de Nivel Alto Tanque 1 (NC)"
   Rectangle "Rectángulo_4" at 444,337 size 33x20
      Appearance <- "Switch de Nivel Bajo Tanque 1 (NO)"
   TextField "Campo de texto_8" at 58,362 size 136x25; Text 'DEL CONTROL'
   GraphicView "Visor de gráficos_5" at 1131,97 size 126x149; Picture "Gráfico_32"
   GraphicView "Visor de gráficos_33" at 1077,115 size 61x29; Picture "Gráfico_16"
   GraphicView "Visor de gráficos_38" at 1157,259 size 56x50; Picture "Gráfico_14"
   GraphicView "Visor de gráficos_39" at 1026,282 size 78x29; Picture "Gráfico_16"
   GraphicView "Visor de gráficos_40" at 1023,82 size 62x64; Picture "Gráfico_23"
   GraphicView "Visor de gráficos_41" at 1099,248 size 62x64; Picture "Gráfico_23"
   GraphicView "Visor de gráficos_42" at 1182,239 size 31x34; Picture "Gráfico_17"
   Button "Botón_11" at 1024,76 size 61x79; TextOff 'Text'
      on Click: InvertBit("v3 llen")
   Button "Botón_12" at 1099,243 size 61x79; TextOff 'Text'
      on Click: InvertBit("v3")
   Circle "Círculo_9" at 1037,43 size 23x23
      Appearance <- "Abrir Valvula Llenado Tanque 3"
   GraphicView "Visor de gráficos_43" at 784,115 size 247x29; Picture "Gráfico_16"
   Circle "Círculo_10" at 1120,323 size 23x23
      Appearance <- "Abrir Valvula Vaciado Tanque 3"
   GraphicView "Visor de gráficos_44" at 739,117 size 53x53; Picture "Gráfico_34"
   GraphicView "Visor de gráficos_45" at 275,51 size 53x149; Picture "Gráfico_35"
   IOField "Campo ES_5" at 248,10 size 96x32; FormatPattern s999999999.999
      ProcessValue <- "temperatura"
   TextField "Campo de texto_9" at 123,12 size 125x25; Text 'Temperatura'
   TextField "Campo de texto_10" at 388,27 size 53x25; Text 'Flujo'
   TextField "Campo de texto_11" at 504,175 size 76x25; Text 'Presion'
   TextField "Campo de texto_12" at 560,10 size 201x25; Text 'Valvula Proporcional'
   TextField "Campo de texto_13" at 366,449 size 159x25; Text 'Velocidad Motor'
   TextField "Campo de texto_14" at 939,171 size 53x25; Text 'Nivel'
   Circle "Círculo_1" at 712,405 size 23x23
      Appearance <- "Abrir Valvula Vaciado Tanque 1"
   Circle "Círculo_2" at 821,405 size 23x23
      Appearance <- "Abrir Valvula Vaciado Tanque 2"
   Circle "Círculo_3" at 700,227 size 23x23
      Appearance <- "Abrir Valvula Llenado Tanque 1"
   Circle "Círculo_4" at 809,225 size 23x23
      Appearance <- "Abrir Valvula Llenado Tanque 2"
   Button "Botón_4" at 1124,490 size 104x70; TextOff 'MANUAL'
      on Click: InvertBit("onproc")
   Button "Botón_14" at 383,511 size 120x84; TextOff 'Text'
      on Click: InvertBit("d7")

screen "fuzzy flujo" 1280x740
   Button "Botón_1" at 915,622 size 250x80; TextOff 'REGRESAR'
      on Click: ActivateScreen("controles flujo", 0)
   Button "Botón_2" at 114,622 size 250x80; TextOff 'PARAMETROS'
      on Click: ActivateScreen("parametros fuzzy flujo", 0)
   Button "Botón_3" at 509,622 size 250x80; TextOff 'TENDENCIAS'
      on Click: ActivateScreen("tendencia fuzzy flujo", 0)
   Button "Botón_5" at 43,193 size 108x49; TextOff 'ON'; TextOn 'OFF'
      on Click: InvertBit("onfuzz")
   TextField "Campo de texto_1" at 33,269 size 99x25; Text 'SETPOINT'
   Circle "Círculo_6" at 167,202 size 32x32
      Appearance <- "onfuzz"
   IOField "Campo ES_1" at 139,262 size 100x40; FormatPattern s999999999.999
      ProcessValue <- "reffuzz"
   GraphicView "Visor de gráficos_7" at 499,243 size 138x216; Picture "Gráfico_11"
   GraphicView "Visor de gráficos_2" at 924,449 size 56x50; Picture "Gráfico_14"
   GraphicView "Visor de gráficos_3" at 554,448 size 53x52; Picture "Gráfico_15"
   GraphicView "Visor de gráficos_4" at 632,290 size 52x29; Picture "Gráfico_16"
   GraphicView "Visor de gráficos_9" at 381,509 size 123x85; Picture "Gráfico_19"
   GraphicView "Visor de gráficos_10" at 388,97 size 61x52; Picture "Gráfico_20"
   GraphicView "Visor de gráficos_11" at 525,67 size 33x57; Picture "Gráfico_21"
   GraphicView "Visor de gráficos_12" at 628,83 size 61x63; Picture "Gráfico_22"
   GraphicView "Visor de gráficos_15" at 681,256 size 62x64; Picture "Gráfico_23"
   GraphicView "Visor de gráficos_17" at 748,469 size 55x58; Picture "Gráfico_24"
   GraphicView "Visor de gráficos_18" at 739,263 size 53x56; Picture "Gráfico_25"
   GraphicView "Visor de gráficos_6" at 790,256 size 62x64; Picture "Gráfico_23"
   GraphicView "Visor de gráficos_19" at 850,290 size 52x29; Picture "Gráfico_16"
   GraphicView "Visor de gráficos_20" at 894,243 size 138x216; Picture "Gráfico_11"
   GraphicView "Visor de gráficos_21" at 603,471 size 92x29; Picture "Gráfico_16"
   GraphicView "Visor de gráficos_22" at 692,437 size 62x64; Picture "Gráfico_23"
   GraphicView "Visor de gráficos_24" at 801,437 size 62x64; Picture "Gráfico_23"
   GraphicView "Visor de gráficos_25" at 861,471 size 67x29; Picture "Gráfico_16"
   GraphicView "Visor de gráficos_1" at 734,515 size 56x50; Picture "Gráfico_14"
   GraphicView "Visor de gráficos_8" at 495,537 size 251x29; Picture "Gráfico_16"
   GraphicView "Visor de gráficos_13" at 306,490 size 54x52; Picture "Gráfico_15"
   GraphicView "Visor de gráficos_14" at 344,513 size 48x29; Picture "Gráfico_16"
   GraphicView "Visor de gráficos_16" at 353,115 size 38x29; Picture "Gráfico_16"
   GraphicView "Visor de gráficos_23" at 445,116 size 187x29; Picture "Gráfico_16"
   GraphicView "Visor de gráficos_26" at 435,221 size 46x68; Picture "Gráfico_26"
   GraphicView "Visor de gráficos_27" at 434,333 size 46x68; Picture "Gráfico_26"
   GraphicView "Visor de gráficos_28" at 462,279 size 45x10; Picture "Gráfico_16"
   GraphicView "Visor de gráficos_29" at 463,391 size 45x10; Picture "Gráfico_16"
   GraphicView "Visor de gráficos_30" at 304,155 size 31x344; Picture "Gráfico_17"
   GraphicView "Visor de gráficos_31" at 307,117 size 52x48; Picture "Gráfico_27"
   GraphicView "Visor de gráficos_32" at 683,116 size 60x29; Picture "Gráfico_16"
   GraphicView "Visor de gráficos_34" at 750,153 size 31x120; Picture "Gráfico_17"
   Circle "Círculo_1" at 712,405 size 23x23
      Appearance <- "v1vac"
   Circle "Círculo_2" at 821,405 size 23x23
      Appearance <- "v2vac"
   Circle "Círculo_3" at 700,227 size 23x23
      Appearance <- "v1llen"
   Circle "Círculo_4" at 809,225 size 23x23
      Appearance <- "v2llen"
   Bar "Barra_1" at 900,275 size 131x145; MinimumValue 0; MaximumValue 27000
      ProcessValue <- "Nivel tanque"
   GraphicView "Visor de gráficos_35" at 930,200 size 75x76; Picture "Gráfico_28"
   Circle "Círculo_5" at 647,144 size 23x23
      Appearance <- "d7"
   GraphicView "Visor de gráficos_37" at 282,217 size 80x80; Picture "Gráfico_30"
   Circle "Círculo_7" at 374,241 size 23x23
      Appearance <- "Activar Unidad Enfriadora"
   Circle "Círculo_8" at 379,403 size 23x23
      Appearance <- "Activar Unidad Calefactora"
   GraphicView "Visor de gráficos_36" at 282,365 size 80x80; Picture "Gráfico_31"
   Rectangle "Rectángulo_2" at 444,225 size 33x20
      Appearance <- "Switch de Nivel Alto Tanque 1 (NC)"
   Rectangle "Rectángulo_4" at 444,337 size 33x20
      Appearance <- "Switch de Nivel Bajo Tanque 1 (NO)"
   GraphicView "Visor de gráficos_5" at 1131,97 size 126x149; Picture "Gráfico_32"
   GraphicView "Visor de gráficos_33" at 1077,115 size 61x29; Picture "Gráfico_16"
   GraphicView "Visor de gráficos_38" at 1157,259 size 56x50; Picture "Gráfico_14"
   GraphicView "Visor de gráficos_39" at 1026,282 size 78x29; Picture "Gráfico_16"
   GraphicView "Visor de gráficos_40" at 1023,82 size 62x64; Picture "Gráfico_23"
   GraphicView "Visor de gráficos_41" at 1099,248 size 62x64; Picture "Gráfico_23"
   GraphicView "Visor de gráficos_42" at 1182,239 size 31x34; Picture "Gráfico_17"
   Circle "Círculo_9" at 1037,43 size 23x23
      Appearance <- "Abrir Valvula Llenado Tanque 3"
   GraphicView "Visor de gráficos_43" at 784,115 size 247x29; Picture "Gráfico_16"
   Circle "Círculo_10" at 1120,323 size 23x23
      Appearance <- "Abrir Valvula Vaciado Tanque 3"
   GraphicView "Visor de gráficos_44" at 739,117 size 53x53; Picture "Gráfico_34"
   GraphicView "Visor de gráficos_45" at 275,51 size 53x149; Picture "Gráfico_35"
   TextField "Campo de texto_9" at 123,12 size 125x25; Text 'Temperatura'
   TextField "Campo de texto_10" at 388,27 size 53x25; Text 'Flujo'
   TextField "Campo de texto_11" at 504,175 size 76x25; Text 'Presion'
   TextField "Campo de texto_12" at 560,10 size 201x25; Text 'Valvula Proporcional'
   TextField "Campo de texto_13" at 366,449 size 159x25; Text 'Velocidad Motor'
   TextField "Campo de texto_14" at 939,171 size 53x25; Text 'Nivel'
   IOField "Campo ES_3" at 249,15 size 96x32; FormatPattern s999999999.999
      ProcessValue <- "temperatura"
   IOField "Campo ES_4" at 371,58 size 96x32; FormatPattern s999999999.999
      ProcessValue <- "flujo"
   IOField "Campo ES_5" at 611,41 size 96x32; FormatPattern s99999
      ProcessValue <- "valvula"
   IOField "Campo ES_6" at 496,147 size 96x32; FormatPattern s999999999.999
      ProcessValue <- "presion"
   IOField "Campo ES_7" at 393,477 size 96x32; FormatPattern s99999
      ProcessValue <- "bomba"
   Button "Botón_6" at 1024,77 size 61x79; TextOff 'Text'
      on Click: InvertBit("v3 llen")
   Button "Botón_7" at 1101,244 size 61x79; TextOff 'Text'
      on Click: InvertBit("v3")
   Button "Botón_8" at 791,250 size 61x79; TextOff 'Text'
      on Click: InvertBit("v2llen")
   Button "Botón_9" at 681,252 size 61x79; TextOff 'Text'
      on Click: InvertBit("v1llen")
   Button "Botón_10" at 695,431 size 61x79; TextOff 'Text'
      on Click: InvertBit("v1vac")
   Button "Botón_11" at 802,431 size 61x79; TextOff 'Text'
      on Click: InvertBit("v2vac")
   Button "Botón_12" at 282,216 size 80x80; TextOff 'Text'
      on Click: InvertBit("enfriadora")
   Button "Botón_13" at 281,366 size 80x80; TextOff 'Text'
      on Click: InvertBit("calefactora")
   TextField "Campo de texto_6" at 41,91 size 191x25; Text 'CONTROL DE FLUJO'
   TextField "Campo de texto_8" at 103,116 size 66x25; Text 'FUZZY'
   TextField "Campo de texto_2" at 69,333 size 133x25; Text 'PARAMETROS'
   TextField "Campo de texto_4" at 37,373 size 109x25; Text 'NEGATIVO'
   TextField "Campo de texto_5" at 78,424 size 55x25; Text 'CERO'
   TextField "Campo de texto_3" at 42,483 size 98x25; Text 'POSITIVO'
   IOField "Campo ES_2" at 138,366 size 100x40; FormatPattern s999999999.999
      ProcessValue <- "NEG_FUZZ"
   IOField "Campo ES_8" at 138,417 size 100x40; FormatPattern s999999999.999
      ProcessValue <- "CERO_FUZ"
   IOField "Campo ES_9" at 138,476 size 100x40; FormatPattern s999999999.999
      ProcessValue <- "POS_FUZZ"
   TextField "Campo de texto_7" at 34,533 size 106x25; Text 'VARIADOR'
   IOField "Campo ES_10" at 138,526 size 100x40; FormatPattern s999999999.999
      ProcessValue <- "VARIADORFUZZ"
   Button "Botón_4" at 1124,490 size 104x70; TextOff 'MANUAL'
      on Click: InvertBit("onproc")
   Button "Botón_14" at 383,511 size 120x84; TextOff 'Text'
      on Click: InvertBit("d7")

screen "lgr presion" 1280x740
   Button "Botón_1" at 792,623 size 250x80; TextOff 'REGRESAR'
      on Click: ActivateScreen("controles presion", 0)
   Button "Botón_3" at 185,623 size 250x80; TextOff 'TENDENCIAS'
      on Click: ActivateScreen("tendencia lgr presion", 0)
   Button "Botón_5" at 48,198 size 108x49; TextOff 'ON'
      on Click: InvertBit("onlgr")
   Circle "Círculo_5" at 177,209 size 35x35
      Appearance <- "onlgr"
   TextField "Campo de texto_1" at 41,278 size 99x25; Text 'SETPOINT'
   TextField "Campo de texto_2" at 75,333 size 135x25; Text 'CONSTANTES'
   TextField "Campo de texto_3" at 58,412 size 43x25; Text 'KP:'
   TextField "Campo de texto_4" at 59,471 size 34x25; Text 'KI:'
   TextField "Campo de texto_5" at 61,531 size 39x25; Text 'KD:'
   IOField "Campo ES_1" at 140,272 size 100x40; FormatPattern s999999999.999
      ProcessValue <- "reflgr"
   TextField "Campo de texto_6" at 42,85 size 216x25; Text 'CONTROL DE PRESION'
   GraphicView "Visor de gráficos_7" at 499,243 size 138x216; Picture "Gráfico_11"
   GraphicView "Visor de gráficos_2" at 924,449 size 56x50; Picture "Gráfico_14"
   GraphicView "Visor de gráficos_3" at 554,448 size 53x52; Picture "Gráfico_15"
   GraphicView "Visor de gráficos_4" at 632,290 size 52x29; Picture "Gráfico_16"
   GraphicView "Visor de gráficos_9" at 381,509 size 123x85; Picture "Gráfico_19"
   GraphicView "Visor de gráficos_10" at 388,97 size 61x52; Picture "Gráfico_20"
   GraphicView "Visor de gráficos_11" at 525,67 size 33x57; Picture "Gráfico_21"
   GraphicView "Visor de gráficos_12" at 628,83 size 61x63; Picture "Gráfico_22"
   GraphicView "Visor de gráficos_15" at 681,256 size 62x64; Picture "Gráfico_23"
   GraphicView "Visor de gráficos_17" at 748,469 size 55x58; Picture "Gráfico_24"
   GraphicView "Visor de gráficos_18" at 739,263 size 53x56; Picture "Gráfico_25"
   GraphicView "Visor de gráficos_6" at 790,256 size 62x64; Picture "Gráfico_23"
   GraphicView "Visor de gráficos_19" at 850,290 size 52x29; Picture "Gráfico_16"
   GraphicView "Visor de gráficos_20" at 894,243 size 138x216; Picture "Gráfico_11"
   GraphicView "Visor de gráficos_21" at 603,471 size 92x29; Picture "Gráfico_16"
   GraphicView "Visor de gráficos_22" at 692,437 size 62x64; Picture "Gráfico_23"
   GraphicView "Visor de gráficos_24" at 801,437 size 62x64; Picture "Gráfico_23"
   GraphicView "Visor de gráficos_25" at 861,471 size 67x29; Picture "Gráfico_16"
   GraphicView "Visor de gráficos_1" at 734,515 size 56x50; Picture "Gráfico_14"
   GraphicView "Visor de gráficos_8" at 495,537 size 251x29; Picture "Gráfico_16"
   GraphicView "Visor de gráficos_13" at 306,490 size 54x52; Picture "Gráfico_15"
   GraphicView "Visor de gráficos_14" at 344,513 size 48x29; Picture "Gráfico_16"
   GraphicView "Visor de gráficos_16" at 353,115 size 38x29; Picture "Gráfico_16"
   GraphicView "Visor de gráficos_23" at 445,116 size 187x29; Picture "Gráfico_16"
   GraphicView "Visor de gráficos_26" at 435,221 size 46x68; Picture "Gráfico_26"
   GraphicView "Visor de gráficos_27" at 434,333 size 46x68; Picture "Gráfico_26"
   GraphicView "Visor de gráficos_28" at 462,279 size 45x10; Picture "Gráfico_16"
   GraphicView "Visor de gráficos_29" at 463,391 size 45x10; Picture "Gráfico_16"
   GraphicView "Visor de gráficos_30" at 304,155 size 31x344; Picture "Gráfico_17"
   GraphicView "Visor de gráficos_31" at 307,117 size 52x48; Picture "Gráfico_27"
   GraphicView "Visor de gráficos_32" at 683,116 size 60x29; Picture "Gráfico_16"
   GraphicView "Visor de gráficos_34" at 750,153 size 31x120; Picture "Gráfico_17"
   Bar "Barra_1" at 900,275 size 131x145; MinimumValue 0; MaximumValue 27000
      ProcessValue <- "Nivel tanque"
   GraphicView "Visor de gráficos_35" at 930,200 size 75x76; Picture "Gráfico_28"
   Circle "Círculo_6" at 647,144 size 23x23
      Appearance <- "d7"
   GraphicView "Visor de gráficos_37" at 282,217 size 80x80; Picture "Gráfico_30"
   Circle "Círculo_7" at 374,241 size 23x23
      Appearance <- "Activar Unidad Enfriadora"
   Circle "Círculo_8" at 379,403 size 23x23
      Appearance <- "Activar Unidad Calefactora"
   GraphicView "Visor de gráficos_36" at 282,365 size 80x80; Picture "Gráfico_31"
   Rectangle "Rectángulo_3" at 444,225 size 33x20
      Appearance <- "Switch de Nivel Alto Tanque 1 (NC)"
   Rectangle "Rectángulo_4" at 444,337 size 33x20
      Appearance <- "Switch de Nivel Bajo Tanque 1 (NO)"
   GraphicView "Visor de gráficos_5" at 1131,97 size 126x149; Picture "Gráfico_32"
   GraphicView "Visor de gráficos_33" at 1077,115 size 61x29; Picture "Gráfico_16"
   GraphicView "Visor de gráficos_38" at 1157,259 size 56x50; Picture "Gráfico_14"
   GraphicView "Visor de gráficos_39" at 1026,282 size 78x29; Picture "Gráfico_16"
   GraphicView "Visor de gráficos_40" at 1023,82 size 62x64; Picture "Gráfico_23"
   GraphicView "Visor de gráficos_41" at 1099,248 size 62x64; Picture "Gráfico_23"
   GraphicView "Visor de gráficos_42" at 1182,239 size 31x34; Picture "Gráfico_17"
   Circle "Círculo_9" at 1037,43 size 23x23
      Appearance <- "Abrir Valvula Llenado Tanque 3"
   GraphicView "Visor de gráficos_43" at 784,115 size 247x29; Picture "Gráfico_16"
   Circle "Círculo_10" at 1120,323 size 23x23
      Appearance <- "Abrir Valvula Vaciado Tanque 3"
   GraphicView "Visor de gráficos_44" at 739,117 size 53x53; Picture "Gráfico_34"
   GraphicView "Visor de gráficos_45" at 275,51 size 53x149; Picture "Gráfico_35"
   TextField "Campo de texto_9" at 123,12 size 125x25; Text 'Temperatura'
   TextField "Campo de texto_10" at 388,27 size 53x25; Text 'Flujo'
   TextField "Campo de texto_11" at 504,175 size 76x25; Text 'Presion'
   TextField "Campo de texto_12" at 560,10 size 201x25; Text 'Valvula Proporcional'
   TextField "Campo de texto_13" at 366,449 size 159x25; Text 'Velocidad Motor'
   TextField "Campo de texto_14" at 939,171 size 53x25; Text 'Nivel'
   IOField "Campo ES_3" at 613,42 size 96x32; FormatPattern s99999
      ProcessValue <- "valvula"
   IOField "Campo ES_4" at 492,145 size 96x32; FormatPattern s999999999.999
      ProcessValue <- "presion"
   IOField "Campo ES_5" at 379,56 size 96x32; FormatPattern s999999999.999
      ProcessValue <- "flujo"
   IOField "Campo ES_6" at 243,11 size 96x32; FormatPattern s999999999.999
      ProcessValue <- "temperatura"
   IOField "Campo ES_7" at 385,475 size 96x32; FormatPattern s99999
      ProcessValue <- "bomba"
   Button "Botón_6" at 680,251 size 61x79; TextOff 'Text'
      on Click: InvertBit("v1llen")
   Button "Botón_7" at 791,251 size 61x79; TextOff 'Text'
      on Click: InvertBit("v2llen")
   Button "Botón_8" at 1099,242 size 61x79; TextOff 'Text'
      on Click: InvertBit("v3")
   Button "Botón_9" at 1024,77 size 61x79; TextOff 'Text'
      on Click: InvertBit("v3 llen")
   Button "Botón_10" at 803,434 size 61x79; TextOff 'Text'
      on Click: InvertBit("v2vac")
   Button "Botón_11" at 694,431 size 61x79; TextOff 'Text'
      on Click: InvertBit("v1vac")
   Button "Botón_12" at 280,364 size 80x80; TextOff 'Text'
      on Click: InvertBit("calefactora")
   Button "Botón_13" at 282,217 size 80x80; TextOff 'Text'
      on Click: InvertBit("enfriadora")
   TextField "Campo de texto_7" at 72,357 size 142x25; Text 'DEL CONTROL'
   IOField "Campo ES_2" at 112,402 size 100x40; FormatPattern s999999999.999
      ProcessValue <- "kp_lgr"
   IOField "Campo ES_8" at 112,463 size 100x40; FormatPattern s999999999.999
      ProcessValue <- "ki_lgr"
   IOField "Campo ES_9" at 113,523 size 100x40; FormatPattern s999999999.999
      ProcessValue <- "kd_lgr"
   TextField "Campo de texto_8" at 36,110 size 238x25; Text 'LUGAR GEOMETRICO DE'
   TextField "Campo de texto_15" at 89,132 size 117x25; Text 'LAS RAICES'
   Circle "Círculo_1" at 712,405 size 23x23
      Appearance <- "Abrir Valvula Vaciado Tanque 1"
   Circle "Círculo_2" at 821,405 size 23x23
      Appearance <- "Abrir Valvula Vaciado Tanque 2"
   Circle "Círculo_3" at 700,227 size 23x23
      Appearance <- "Abrir Valvula Llenado Tanque 1"
   Circle "Círculo_4" at 809,225 size 23x23
      Appearance <- "Abrir Valvula Llenado Tanque 2"
   Button "Botón_4" at 1124,490 size 104x70; TextOff 'MANUAL'
      on Click: InvertBit("onproc")
   Button "Botón_14" at 383,511 size 120x84; TextOff 'Text'
      on Click: InvertBit("d7")

screen "predictor smith flujo" 1280x740
   Button "Botón_1" at 833,624 size 250x80; TextOff 'REGRESAR'
      on Click: ActivateScreen("controles flujo", 0)
   Button "Botón_3" at 235,626 size 250x80; TextOff 'TENDENCIAS'
      on Click: ActivateScreen("tendencia smith flujo", 0)
   Button "Botón_5" at 38,194 size 108x49; TextOff 'ON'
      on Click: InvertBit("onsmith")
   IOField "Campo ES_1" at 136,259 size 100x40; FormatPattern s999999999.999
      ProcessValue <- "refsm"
   Circle "Círculo_5" at 168,199 size 39x39
      Appearance <- "onsmith"
   TextField "Campo de texto_1" at 28,264 size 99x25; Text 'SETPOINT'
   GraphicView "Visor de gráficos_7" at 499,243 size 138x216; Picture "Gráfico_11"
   GraphicView "Visor de gráficos_2" at 924,449 size 56x50; Picture "Gráfico_14"
   GraphicView "Visor de gráficos_3" at 554,448 size 53x52; Picture "Gráfico_15"
   GraphicView "Visor de gráficos_4" at 632,290 size 52x29; Picture "Gráfico_16"
   GraphicView "Visor de gráficos_9" at 381,509 size 123x85; Picture "Gráfico_19"
   GraphicView "Visor de gráficos_10" at 388,97 size 61x52; Picture "Gráfico_20"
   GraphicView "Visor de gráficos_11" at 525,67 size 33x57; Picture "Gráfico_21"
   GraphicView "Visor de gráficos_12" at 628,83 size 61x63; Picture "Gráfico_22"
   GraphicView "Visor de gráficos_15" at 681,256 size 62x64; Picture "Gráfico_23"
   GraphicView "Visor de gráficos_17" at 748,469 size 55x58; Picture "Gráfico_24"
   GraphicView "Visor de gráficos_18" at 739,263 size 53x56; Picture "Gráfico_25"
   GraphicView "Visor de gráficos_6" at 790,256 size 62x64; Picture "Gráfico_23"
   GraphicView "Visor de gráficos_19" at 850,290 size 52x29; Picture "Gráfico_16"
   GraphicView "Visor de gráficos_20" at 894,243 size 138x216; Picture "Gráfico_11"
   GraphicView "Visor de gráficos_21" at 603,471 size 92x29; Picture "Gráfico_16"
   GraphicView "Visor de gráficos_22" at 692,437 size 62x64; Picture "Gráfico_23"
   GraphicView "Visor de gráficos_24" at 801,437 size 62x64; Picture "Gráfico_23"
   GraphicView "Visor de gráficos_25" at 861,471 size 67x29; Picture "Gráfico_16"
   GraphicView "Visor de gráficos_1" at 734,515 size 56x50; Picture "Gráfico_14"
   GraphicView "Visor de gráficos_8" at 495,537 size 251x29; Picture "Gráfico_16"
   GraphicView "Visor de gráficos_13" at 307,490 size 54x52; Picture "Gráfico_15"
   GraphicView "Visor de gráficos_14" at 344,513 size 48x29; Picture "Gráfico_16"
   GraphicView "Visor de gráficos_16" at 353,115 size 38x29; Picture "Gráfico_16"
   GraphicView "Visor de gráficos_23" at 445,116 size 187x29; Picture "Gráfico_16"
   GraphicView "Visor de gráficos_26" at 435,221 size 46x68; Picture "Gráfico_26"
   GraphicView "Visor de gráficos_27" at 434,333 size 46x68; Picture "Gráfico_26"
   GraphicView "Visor de gráficos_28" at 462,279 size 45x10; Picture "Gráfico_16"
   GraphicView "Visor de gráficos_29" at 463,391 size 45x10; Picture "Gráfico_16"
   GraphicView "Visor de gráficos_30" at 306,155 size 31x344; Picture "Gráfico_17"
   GraphicView "Visor de gráficos_31" at 307,117 size 52x48; Picture "Gráfico_27"
   GraphicView "Visor de gráficos_32" at 683,116 size 60x29; Picture "Gráfico_16"
   GraphicView "Visor de gráficos_34" at 750,153 size 31x120; Picture "Gráfico_17"
   Bar "Barra_1" at 900,275 size 131x145; MinimumValue 0; MaximumValue 27000
      ProcessValue <- "Nivel tanque"
   GraphicView "Visor de gráficos_35" at 930,200 size 75x76; Picture "Gráfico_28"
   Circle "Círculo_6" at 647,144 size 23x23
      Appearance <- "d7"
   GraphicView "Visor de gráficos_37" at 282,217 size 80x80; Picture "Gráfico_30"
   Circle "Círculo_7" at 374,241 size 23x23
      Appearance <- "Activar Unidad Enfriadora"
   Circle "Círculo_8" at 379,403 size 23x23
      Appearance <- "Activar Unidad Calefactora"
   GraphicView "Visor de gráficos_36" at 282,365 size 80x80; Picture "Gráfico_31"
   Rectangle "Rectángulo_2" at 444,225 size 33x20
      Appearance <- "Switch de Nivel Alto Tanque 1 (NC)"
   Rectangle "Rectángulo_4" at 444,337 size 33x20
      Appearance <- "Switch de Nivel Bajo Tanque 1 (NO)"
   GraphicView "Visor de gráficos_5" at 1131,97 size 126x149; Picture "Gráfico_32"
   GraphicView "Visor de gráficos_33" at 1077,115 size 61x29; Picture "Gráfico_16"
   GraphicView "Visor de gráficos_38" at 1157,259 size 56x50; Picture "Gráfico_14"
   GraphicView "Visor de gráficos_39" at 1026,282 size 78x29; Picture "Gráfico_16"
   GraphicView "Visor de gráficos_40" at 1023,82 size 62x64; Picture "Gráfico_23"
   GraphicView "Visor de gráficos_41" at 1099,248 size 62x64; Picture "Gráfico_23"
   GraphicView "Visor de gráficos_42" at 1182,239 size 31x34; Picture "Gráfico_17"
   Circle "Círculo_9" at 1037,43 size 23x23
      Appearance <- "Abrir Valvula Llenado Tanque 3"
   GraphicView "Visor de gráficos_43" at 784,115 size 247x29; Picture "Gráfico_16"
   Circle "Círculo_10" at 1120,323 size 23x23
      Appearance <- "Abrir Valvula Vaciado Tanque 3"
   GraphicView "Visor de gráficos_44" at 739,117 size 53x53; Picture "Gráfico_34"
   GraphicView "Visor de gráficos_45" at 275,51 size 53x149; Picture "Gráfico_35"
   TextField "Campo de texto_9" at 123,12 size 125x25; Text 'Temperatura'
   TextField "Campo de texto_10" at 388,27 size 53x25; Text 'Flujo'
   TextField "Campo de texto_11" at 504,175 size 76x25; Text 'Presion'
   TextField "Campo de texto_12" at 560,10 size 201x25; Text 'Valvula Proporcional'
   TextField "Campo de texto_13" at 366,449 size 159x25; Text 'Velocidad Motor'
   TextField "Campo de texto_14" at 939,171 size 53x25; Text 'Nivel'
   IOField "Campo ES_3" at 253,11 size 96x32; FormatPattern s999999999.999
      ProcessValue <- "temperatura"
   IOField "Campo ES_4" at 375,55 size 96x32; FormatPattern s999999999.999
      ProcessValue <- "flujo"
   IOField "Campo ES_5" at 613,44 size 96x32; FormatPattern s99999
      ProcessValue <- "valvula"
   IOField "Campo ES_6" at 492,148 size 96x32; FormatPattern s999999999.999
      ProcessValue <- "presion"
   IOField "Campo ES_7" at 401,475 size 96x32; FormatPattern s99999
      ProcessValue <- "bomba"
   Button "Botón_6" at 1024,77 size 61x79; TextOff 'Text'
      on Click: InvertBit("v3 llen")
   Button "Botón_7" at 681,252 size 61x79; TextOff 'Text'
      on Click: InvertBit("v1llen")
   Button "Botón_8" at 790,252 size 61x79; TextOff 'Text'
      on Click: InvertBit("v2llen")
   Button "Botón_9" at 693,432 size 61x79; TextOff 'Text'
      on Click: InvertBit("v1vac")
   Button "Botón_10" at 801,432 size 61x79; TextOff 'Text'
      on Click: InvertBit("v2vac")
   Button "Botón_11" at 1100,243 size 61x79; TextOff 'Text'
      on Click: InvertBit("v3")
   Button "Botón_12" at 281,217 size 80x80; TextOff 'Text'
      on Click: InvertBit("enfriadora")
   Button "Botón_13" at 283,364 size 80x80; TextOff 'Text'
      on Click: InvertBit("calefactora")
   TextField "Campo de texto_2" at 75,333 size 135x25; Text 'CONSTANTES'
   TextField "Campo de texto_3" at 58,412 size 43x25; Text 'KP:'
   TextField "Campo de texto_4" at 59,471 size 34x25; Text 'KI:'
   TextField "Campo de texto_5" at 61,531 size 39x25; Text 'KD:'
   TextField "Campo de texto_7" at 72,357 size 142x25; Text 'DEL CONTROL'
   IOField "Campo ES_2" at 109,405 size 100x40; FormatPattern s999999999.999
      ProcessValue <- "kp_smith"
   IOField "Campo ES_8" at 109,464 size 100x40; FormatPattern s999999999.999
      ProcessValue <- "ki_smith"
   IOField "Campo ES_9" at 109,524 size 100x40; FormatPattern s999999999.999
      ProcessValue <- "kd_smith"
   TextField "Campo de texto_6" at 45,88 size 191x25; Text 'CONTROL DE FLUJO'
   TextField "Campo de texto_8" at 34,113 size 213x25; Text 'PREDICTOR DE SMITH'
   Circle "Círculo_1" at 712,405 size 23x23
      Appearance <- "Abrir Valvula Vaciado Tanque 1"
   Circle "Círculo_2" at 821,405 size 23x23
      Appearance <- "Abrir Valvula Vaciado Tanque 2"
   Circle "Círculo_3" at 700,227 size 23x23
      Appearance <- "Abrir Valvula Llenado Tanque 1"
   Circle "Círculo_4" at 809,225 size 23x23
      Appearance <- "Abrir Valvula Llenado Tanque 2"
   Button "Botón_4" at 1124,490 size 104x70; TextOff 'MANUAL'
      on Click: InvertBit("onproc")
   Button "Botón_14" at 383,511 size 120x84; TextOff 'Text'
      on Click: InvertBit("d7")

screen "smithant flujo" 1280x740
   Button "Botón_1" at 833,623 size 250x80; TextOff 'REGRESAR'
      on Click: ActivateScreen("controles flujo", 0)
   Button "Botón_3" at 222,623 size 250x80; TextOff 'TENDENCIAS'
      on Click: ActivateScreen("tendencia smithant flujo", 0)
   Button "Botón_5" at 53,196 size 108x49; TextOff 'ON'
      on Click: InvertBit("onsmtant")
   IOField "Campo ES_1" at 143,264 size 100x40; FormatPattern s999999999.999
      ProcessValue <- "refsmtant"
   Circle "Círculo_5" at 186,204 size 34x34
      Appearance <- "onsmtant"
   GraphicView "Visor de gráficos_7" at 499,243 size 138x216; Picture "Gráfico_11"
   GraphicView "Visor de gráficos_2" at 924,449 size 56x50; Picture "Gráfico_14"
   GraphicView "Visor de gráficos_3" at 554,448 size 53x52; Picture "Gráfico_15"
   GraphicView "Visor de gráficos_4" at 632,290 size 52x29; Picture "Gráfico_16"
   GraphicView "Visor de gráficos_9" at 381,509 size 123x85; Picture "Gráfico_19"
   GraphicView "Visor de gráficos_10" at 388,97 size 61x52; Picture "Gráfico_20"
   GraphicView "Visor de gráficos_11" at 525,67 size 33x57; Picture "Gráfico_21"
   GraphicView "Visor de gráficos_12" at 628,83 size 61x63; Picture "Gráfico_22"
   GraphicView "Visor de gráficos_15" at 681,256 size 62x64; Picture "Gráfico_23"
   GraphicView "Visor de gráficos_17" at 748,469 size 55x58; Picture "Gráfico_24"
   GraphicView "Visor de gráficos_18" at 739,263 size 53x56; Picture "Gráfico_25"
   GraphicView "Visor de gráficos_6" at 790,256 size 62x64; Picture "Gráfico_23"
   GraphicView "Visor de gráficos_19" at 850,290 size 52x29; Picture "Gráfico_16"
   GraphicView "Visor de gráficos_20" at 894,243 size 138x216; Picture "Gráfico_11"
   GraphicView "Visor de gráficos_21" at 603,471 size 92x29; Picture "Gráfico_16"
   GraphicView "Visor de gráficos_22" at 692,437 size 62x64; Picture "Gráfico_23"
   GraphicView "Visor de gráficos_24" at 801,437 size 62x64; Picture "Gráfico_23"
   GraphicView "Visor de gráficos_25" at 861,471 size 67x29; Picture "Gráfico_16"
   GraphicView "Visor de gráficos_1" at 734,515 size 56x50; Picture "Gráfico_14"
   GraphicView "Visor de gráficos_8" at 495,537 size 251x29; Picture "Gráfico_16"
   GraphicView "Visor de gráficos_13" at 306,490 size 54x52; Picture "Gráfico_15"
   GraphicView "Visor de gráficos_14" at 344,513 size 48x29; Picture "Gráfico_16"
   GraphicView "Visor de gráficos_16" at 353,115 size 38x29; Picture "Gráfico_16"
   GraphicView "Visor de gráficos_23" at 445,116 size 187x29; Picture "Gráfico_16"
   GraphicView "Visor de gráficos_26" at 435,221 size 46x68; Picture "Gráfico_26"
   GraphicView "Visor de gráficos_27" at 434,333 size 46x68; Picture "Gráfico_26"
   GraphicView "Visor de gráficos_28" at 462,279 size 45x10; Picture "Gráfico_16"
   GraphicView "Visor de gráficos_29" at 463,391 size 45x10; Picture "Gráfico_16"
   GraphicView "Visor de gráficos_30" at 304,155 size 31x344; Picture "Gráfico_17"
   GraphicView "Visor de gráficos_31" at 307,117 size 52x48; Picture "Gráfico_27"
   GraphicView "Visor de gráficos_32" at 683,116 size 60x29; Picture "Gráfico_16"
   GraphicView "Visor de gráficos_34" at 750,153 size 31x120; Picture "Gráfico_17"
   Circle "Círculo_1" at 712,405 size 23x23
      Appearance <- "Abrir Valvula Vaciado Tanque 1"
   Circle "Círculo_2" at 821,405 size 23x23
      Appearance <- "Abrir Valvula Vaciado Tanque 2"
   Circle "Círculo_3" at 700,227 size 23x23
      Appearance <- "Abrir Valvula Llenado Tanque 1"
   Circle "Círculo_4" at 809,225 size 23x23
      Appearance <- "Abrir Valvula Llenado Tanque 2"
   Bar "Barra_1" at 900,275 size 131x145; MinimumValue 0; MaximumValue 27000
      ProcessValue <- "Nivel tanque"
   GraphicView "Visor de gráficos_35" at 930,200 size 75x76; Picture "Gráfico_28"
   Circle "Círculo_6" at 647,144 size 23x23
      Appearance <- "d7"
   GraphicView "Visor de gráficos_37" at 282,217 size 80x80; Picture "Gráfico_30"
   Circle "Círculo_7" at 374,241 size 23x23
      Appearance <- "Activar Unidad Enfriadora"
   Circle "Círculo_8" at 379,403 size 23x23
      Appearance <- "Activar Unidad Calefactora"
   GraphicView "Visor de gráficos_36" at 282,365 size 80x80; Picture "Gráfico_31"
   Rectangle "Rectángulo_2" at 444,225 size 33x20
      Appearance <- "Switch de Nivel Alto Tanque 1 (NC)"
   Rectangle "Rectángulo_4" at 444,337 size 33x20
      Appearance <- "Switch de Nivel Bajo Tanque 1 (NO)"
   GraphicView "Visor de gráficos_5" at 1131,97 size 126x149; Picture "Gráfico_32"
   GraphicView "Visor de gráficos_33" at 1077,115 size 61x29; Picture "Gráfico_16"
   GraphicView "Visor de gráficos_38" at 1157,259 size 56x50; Picture "Gráfico_14"
   GraphicView "Visor de gráficos_39" at 1026,282 size 78x29; Picture "Gráfico_16"
   GraphicView "Visor de gráficos_40" at 1023,82 size 62x64; Picture "Gráfico_23"
   GraphicView "Visor de gráficos_41" at 1099,248 size 62x64; Picture "Gráfico_23"
   GraphicView "Visor de gráficos_42" at 1182,239 size 31x34; Picture "Gráfico_17"
   Circle "Círculo_9" at 1037,43 size 23x23
      Appearance <- "Abrir Valvula Llenado Tanque 3"
   GraphicView "Visor de gráficos_43" at 784,115 size 247x29; Picture "Gráfico_16"
   Circle "Círculo_10" at 1120,323 size 23x23
      Appearance <- "Abrir Valvula Vaciado Tanque 3"
   GraphicView "Visor de gráficos_44" at 739,117 size 53x53; Picture "Gráfico_34"
   GraphicView "Visor de gráficos_45" at 275,51 size 53x149; Picture "Gráfico_35"
   TextField "Campo de texto_9" at 123,12 size 125x25; Text 'Temperatura'
   TextField "Campo de texto_10" at 388,27 size 53x25; Text 'Flujo'
   TextField "Campo de texto_11" at 504,175 size 76x25; Text 'Presion'
   TextField "Campo de texto_12" at 560,10 size 201x25; Text 'Valvula Proporcional'
   TextField "Campo de texto_13" at 366,449 size 159x25; Text 'Velocidad Motor'
   TextField "Campo de texto_14" at 939,171 size 53x25; Text 'Nivel'
   IOField "Campo ES_3" at 250,13 size 96x32; FormatPattern s999999999.999
      ProcessValue <- "temperatura"
   IOField "Campo ES_4" at 364,60 size 96x32; FormatPattern s999999999.999
      ProcessValue <- "flujo"
   IOField "Campo ES_5" at 613,41 size 96x32; FormatPattern s99999
      ProcessValue <- "valvula"
   IOField "Campo ES_6" at 493,146 size 96x32; FormatPattern s999999999.999
      ProcessValue <- "presion"
   IOField "Campo ES_7" at 405,476 size 96x32; FormatPattern s99999
      ProcessValue <- "bomba"
   Button "Botón_6" at 1024,76 size 61x79; TextOff 'Text'
      on Click: InvertBit("v3 llen")
   Button "Botón_7" at 1100,244 size 61x79; TextOff 'Text'
      on Click: InvertBit("v3")
   Button "Botón_8" at 682,251 size 61x79; TextOff 'Text'
      on Click: InvertBit("v1llen")
   Button "Botón_9" at 791,251 size 61x79; TextOff 'Text'
      on Click: InvertBit("v2llen")
   Button "Botón_10" at 693,432 size 61x79; TextOff 'Text'
      on Click: InvertBit("v1vac")
   Button "Botón_11" at 802,430 size 61x79; TextOff 'Text'
      on Click: InvertBit("v2vac")
   Button "Botón_12" at 281,219 size 80x80; TextOff 'Text'
      on Click: InvertBit("enfriadora")
   Button "Botón_13" at 280,365 size 80x80; TextOff 'Text'
      on Click: InvertBit("calefactora")
   TextField "Campo de texto_6" at 45,80 size 191x25; Text 'CONTROL DE FLUJO'
   TextField "Campo de texto_8" at 34,105 size 213x25; Text 'PREDICTOR DE SMITH'
   TextField "Campo de texto_2" at 75,333 size 135x25; Text 'CONSTANTES'
   TextField "Campo de texto_3" at 58,412 size 43x25; Text 'KP:'
   TextField "Campo de texto_4" at 59,471 size 34x25; Text 'KI:'
   TextField "Campo de texto_5" at 61,531 size 39x25; Text 'KD:'
   TextField "Campo de texto_7" at 72,357 size 142x25; Text 'DEL CONTROL'
   IOField "Campo ES_2" at 110,405 size 100x40; FormatPattern s999999999.999
      ProcessValue <- "kp_smitant"
   IOField "Campo ES_8" at 110,464 size 100x40; FormatPattern s999999999.999
      ProcessValue <- "ki_smitant"
   IOField "Campo ES_10" at 110,524 size 100x40; FormatPattern s999999999.999
      ProcessValue <- "kd_smitant"
   TextField "Campo de texto_1" at 42,271 size 99x25; Text 'SETPOINT'
   TextField "Campo de texto_15" at 69,131 size 144x25; Text 'ANTICIPATIVO'
   Button "Botón_4" at 1124,490 size 104x70; TextOff 'MANUAL'
      on Click: InvertBit("onproc")
   Button "Botón_14" at 383,511 size 120x84; TextOff 'Text'
      on Click: InvertBit("d7")

screen "tendencia lgr presion" 1280x740
   Button "Botón_1" at 535,607 size 300x80; TextOff 'REGRESAR'
      on Click: ActivateScreen("lgr presion", 0)
   TrendView "Visor de curvas_1" at 164,122 size 991x414
   TextField "Campo de texto_1" at 276,63 size 761x39; Text 'TENDENCIA DEL CONTROL DE PRESION POR PID'

screen "tendencia on-off temperatura" 1280x740
   Button "Botón_1" at 509,615 size 300x80; TextOff 'REGRESAR'
      on Click: ActivateScreen("on-off temperatura", 0)
   TrendView "Visor de curvas_1" at 135,149 size 1030x365
   TextField "Campo de texto_1" at 300,69 size 718x39; Text 'TENDENCIA DEL CONTROL DE TEMPERATURA'

screen "tendencia fuzzy flujo" 1280x740
   TextField "Campo de texto_1" at 311,49 size 692x39; Text 'TENDENCIA DEL CONTROL DE FLUJO FUZZY'
   Button "Botón_1" at 509,611 size 300x80; TextOff 'REGRESAR'
      on Click: ActivateScreen("fuzzy flujo", 0)
   TrendView "Visor de curvas_1" at 115,101 size 1088x445

screen "tendencia smith flujo" 1280x740
   TextField "Campo de texto_1" at 300,49 size 697x39; Text 'TENDENCIA DEL CONTROL DE FLUJO SMITH'
   Button "Botón_1" at 509,615 size 300x80; TextOff 'REGRESAR'
      on Click: ActivateScreen("predictor smith flujo", 0)
   TrendView "Visor de curvas_1" at 164,116 size 996x416

screen "tendencia smithant flujo" 1280x740
   TextField "Campo de texto_1" at 190,69 size 939x39; Text 'TENDENCIA DEL CONTROL DE FLUJO SMITH ANTICIPATIVO'
   TrendView "Visor de curvas_1" at 130,140 size 1058x392
   Button "Botón_1" at 509,609 size 300x80; TextOff 'REGRESAR'
      on Click: ActivateScreen("smithant flujo", 0)

screen "manual" 1280x740
   Button "Botón_1" at 940,586 size 258x86; TextOff 'regresar'
      on Click: ActivateScreen("controles flujo", 0)
   Button "Botón_2" at 284,202 size 132x82; TextOff 'V1 LLEN'
      on Click: InvertBit("v1llen")
   Button "Botón_3" at 286,326 size 130x98; TextOff 'V1 VAC'
      on Click: InvertBit("v1vac")
   Button "Botón_4" at 696,208 size 152x74; TextOff 'V2 LLEN'
      on Click: InvertBit("v2llen")
   Button "Botón_5" at 698,326 size 146x88; TextOff 'V2 VAC'
      on Click: InvertBit("v2vac")
   Button "Botón_6" at 466,456 size 170x102; TextOff 'V3'
      on Click: InvertBit("v3")
   Button "Botón_7" at 86,604 size 238x66; TextOff 'ON PROCESO'
      on Click: InvertBit("onproc")
   Button "Botón_8" at 448,70 size 222x76; TextOff 'VALVULA PRINCIPAL'
      on Click: InvertBit("d7")
   TextField "Campo de texto_1" at 970,94 size 248x25; Text 'VALVULA PROPORCIONAL'
   TextField "Campo de texto_2" at 970,226 size 222x25; Text 'VELOCIDAD VARIADOR'
   IOField "Campo ES_1" at 976,134 size 218x68; FormatPattern s99999
      ProcessValue <- "valvula"
   IOField "Campo ES_2" at 980,278 size 212x60; FormatPattern s99999
      ProcessValue <- "bomba"

screen "tendencia sintonizacion flujo" 1280x740
   TrendView "Visor de curvas_1" at 200,122 size 918x394
   Button "Botón_1" at 509,614 size 300x80; TextOff 'REGRESAR'
      on Click: ActivateScreen("sintonizacion flujo", 0)
   TextField "Campo de texto_1" at 234,48 size 927x39; Text 'TENDENCIA DEL CONTROL DE FLUJO POR SINTONIZACION'

screen "INFO" 1280x740
   Button "Botón_1" at 1002,588 size 192x102; TextOff 'REGRESAR'
      on Click: ActivateScreen("controles flujo", 0)
   GraphicView "Visor de gráficos_1" at 192,75 size 400x625; Picture "PLANTAPRES"
   Button "Botón_4" at 750,326 size 174x96; TextOff 'PROBLEMATICA'
      on Click: ActivateScreen("PROBLEMATICA", 0)
   Button "Botón_5" at 750,448 size 174x90; TextOff 'RESUMEN'
      on Click: ActivateScreen("RESUMEN", 0)
   Button "Botón_6" at 754,562 size 170x96; TextOff 'DESCRIPCION'
      on Click: ActivateScreen("DESCRIPCION", 0)
   TextField "HmiScreenItemData" at 10,0 size 1270x79; Text '"TÉCNICA DE CONTROL Y SUPERVISION EN EL MODULO DE PROCESOS"'
   Button "Botón_2" at 744,94 size 188x88; TextOff 'P&ID'
      on Click: ActivateScreen("P&ID", 0)
   Button "Botón_3" at 748,206 size 182x82; TextOff 'ARQUITECTURA'
      on Click: ActivateScreen("ARQUIT", 0)

screen "P&ID" 1280x740
   GraphicView "Visor de gráficos_1" at 110,0 size 1021x689; Picture "P&ID"
   Button "Botón_1" at 1136,646 size 132x76; TextOff 'REGRESAR'
      on Click: ActivateScreen("INFO", 0)

screen "ARQUIT" 1280x740
   GraphicView "Visor de gráficos_1" at 136,0 size 1013x705; Picture "ARQUITECTURA"
   Button "Botón_1" at 1150,658 size 116x56; TextOff 'REGRESAR'
      on Click: ActivateScreen("INFO", 0)

screen "PROBLEMATICA" 1280x740
   TextField "HmiScreenItemData" at 0,8 size 1270x79; Text '"TÉCNICA DE CONTROL Y SUPERVISION EN EL MODULO DE PROCESOS"'
   TextField "HmiScreenItemData_1" at 8,52 size 1270x77; Text '"AUTOMATIZACION DE PROCESOS"'
   TextField "HmiScreenItemData_2" at 8,96 size 1270x71; Text '2016'
   Button "Botón_1" at 964,604 size 268x96; TextOff 'REGRESAR'
      on Click: ActivateScreen("INFO", 0)
   GraphicView "Visor de gráficos_1" at 231,221 size 863x268; Picture "HH"

screen "RESUMEN" 1280x740
   Button "Botón_1" at 1006,582 size 212x110; TextOff 'REGRESAR'
      on Click: ActivateScreen("INFO", 0)
   TextField "HmiScreenItemData" at 0,8 size 1270x79; Text '"TÉCNICA DE CONTROL Y SUPERVISION EN EL MODULO DE PROCESOS"'
   TextField "HmiScreenItemData_1" at 8,52 size 1270x77; Text '"AUTOMATIZACION DE PROCESOS"'
   TextField "HmiScreenItemData_2" at 8,96 size 1270x71; Text '2016'
   GraphicView "Visor de gráficos_1" at 230,212 size 895x283; Picture "RESUMEN"

screen "DESCRIPCION" 1280x740
   TextField "HmiScreenItemData" at 0,8 size 1270x79; Text '"TÉCNICA DE CONTROL Y SUPERVISION EN EL MODULO DE PROCESOS"'
   TextField "HmiScreenItemData_1" at 8,52 size 1270x77; Text '"AUTOMATIZACION DE PROCESOS"'
   TextField "HmiScreenItemData_2" at 8,96 size 1270x71; Text '2016'
   Button "Botón_1" at 1012,594 size 238x114; TextOff 'REGRESAR'
      on Click: ActivateScreen("INFO", 0)
   GraphicView "Visor de gráficos_1" at 220,196 size 895x310; Picture "DESCRP"

screen "on-off temperatura" 1280x740
   TextField "Campo de texto_1" at 68,273 size 140x32; Text 'SETPOINT'
   TextField "Campo de texto_2" at 43,405 size 191x32; Text 'TEMPERATURA'
   Button "Botón_1" at 48,183 size 108x49; TextOff 'ON'
      on Click: InvertBit("on_temp")
   IOField "Campo ES_1" at 51,313 size 176x58; FormatPattern s999999999.999
      ProcessValue <- "REFTEMP"
   IOField "Campo ES_2" at 51,484 size 176x58; FormatPattern s999999999.999
      ProcessValue <- "temperatura"
   Button "Botón_2" at 732,622 size 300x80; TextOff 'REGRESAR'
      on Click: ActivateScreen("controles temperatura", 0)
   GraphicView "Visor de gráficos_7" at 499,243 size 138x216; Picture "Gráfico_11"
   GraphicView "Visor de gráficos_2" at 924,449 size 56x50; Picture "Gráfico_14"
   GraphicView "Visor de gráficos_3" at 554,448 size 53x52; Picture "Gráfico_15"
   GraphicView "Visor de gráficos_4" at 632,290 size 52x29; Picture "Gráfico_16"
   GraphicView "Visor de gráficos_9" at 381,509 size 123x85; Picture "Gráfico_19"
   GraphicView "Visor de gráficos_10" at 388,97 size 61x52; Picture "Gráfico_20"
   GraphicView "Visor de gráficos_11" at 525,67 size 33x57; Picture "Gráfico_21"
   GraphicView "Visor de gráficos_12" at 628,83 size 61x63; Picture "Gráfico_22"
   GraphicView "Visor de gráficos_15" at 681,256 size 62x64; Picture "Gráfico_23"
   GraphicView "Visor de gráficos_17" at 748,469 size 55x58; Picture "Gráfico_24"
   GraphicView "Visor de gráficos_18" at 739,263 size 53x56; Picture "Gráfico_25"
   GraphicView "Visor de gráficos_6" at 790,256 size 62x64; Picture "Gráfico_23"
   GraphicView "Visor de gráficos_19" at 850,290 size 52x29; Picture "Gráfico_16"
   GraphicView "Visor de gráficos_20" at 894,243 size 138x216; Picture "Gráfico_11"
   GraphicView "Visor de gráficos_21" at 603,471 size 92x29; Picture "Gráfico_16"
   GraphicView "Visor de gráficos_22" at 692,437 size 62x64; Picture "Gráfico_23"
   GraphicView "Visor de gráficos_24" at 801,437 size 62x64; Picture "Gráfico_23"
   GraphicView "Visor de gráficos_25" at 861,471 size 67x29; Picture "Gráfico_16"
   GraphicView "Visor de gráficos_1" at 734,515 size 56x50; Picture "Gráfico_14"
   GraphicView "Visor de gráficos_8" at 495,537 size 251x29; Picture "Gráfico_16"
   GraphicView "Visor de gráficos_13" at 306,490 size 54x52; Picture "Gráfico_15"
   GraphicView "Visor de gráficos_14" at 344,513 size 48x29; Picture "Gráfico_16"
   GraphicView "Visor de gráficos_16" at 353,115 size 38x29; Picture "Gráfico_16"
   GraphicView "Visor de gráficos_23" at 445,116 size 187x29; Picture "Gráfico_16"
   GraphicView "Visor de gráficos_26" at 435,221 size 46x68; Picture "Gráfico_26"
   GraphicView "Visor de gráficos_27" at 434,333 size 46x68; Picture "Gráfico_26"
   GraphicView "Visor de gráficos_28" at 462,279 size 45x10; Picture "Gráfico_16"
   GraphicView "Visor de gráficos_29" at 463,391 size 45x10; Picture "Gráfico_16"
   GraphicView "Visor de gráficos_30" at 304,155 size 31x344; Picture "Gráfico_17"
   GraphicView "Visor de gráficos_31" at 307,117 size 52x48; Picture "Gráfico_27"
   GraphicView "Visor de gráficos_32" at 683,116 size 60x29; Picture "Gráfico_16"
   GraphicView "Visor de gráficos_34" at 750,153 size 31x120; Picture "Gráfico_17"
   Bar "Barra_1" at 900,275 size 131x145; MinimumValue 0; MaximumValue 27000
      ProcessValue <- "Nivel tanque"
   GraphicView "Visor de gráficos_35" at 930,200 size 75x76; Picture "Gráfico_28"
   Circle "Círculo_6" at 647,144 size 23x23
      Appearance <- "d7"
   GraphicView "Visor de gráficos_37" at 282,217 size 80x80; Picture "Gráfico_30"
   Circle "Círculo_7" at 374,241 size 23x23
      Appearance <- "Activar Unidad Enfriadora"
   Circle "Círculo_8" at 379,403 size 23x23
      Appearance <- "Activar Unidad Calefactora"
   GraphicView "Visor de gráficos_36" at 282,365 size 80x80; Picture "Gráfico_31"
   Rectangle "Rectángulo_2" at 444,225 size 33x20
      Appearance <- "Switch de Nivel Alto Tanque 1 (NC)"
   Rectangle "Rectángulo_4" at 444,337 size 33x20
      Appearance <- "Switch de Nivel Bajo Tanque 1 (NO)"
   GraphicView "Visor de gráficos_5" at 1131,97 size 126x149; Picture "Gráfico_32"
   GraphicView "Visor de gráficos_33" at 1077,115 size 61x29; Picture "Gráfico_16"
   GraphicView "Visor de gráficos_38" at 1157,259 size 56x50; Picture "Gráfico_14"
   GraphicView "Visor de gráficos_39" at 1026,282 size 78x29; Picture "Gráfico_16"
   GraphicView "Visor de gráficos_40" at 1023,82 size 62x64; Picture "Gráfico_23"
   GraphicView "Visor de gráficos_41" at 1099,248 size 62x64; Picture "Gráfico_23"
   GraphicView "Visor de gráficos_42" at 1182,239 size 31x34; Picture "Gráfico_17"
   Circle "Círculo_9" at 1037,43 size 23x23
      Appearance <- "Abrir Valvula Llenado Tanque 3"
   GraphicView "Visor de gráficos_43" at 784,115 size 247x29; Picture "Gráfico_16"
   Circle "Círculo_10" at 1120,323 size 23x23
      Appearance <- "Abrir Valvula Vaciado Tanque 3"
   GraphicView "Visor de gráficos_44" at 739,117 size 53x53; Picture "Gráfico_34"
   GraphicView "Visor de gráficos_45" at 275,51 size 53x149; Picture "Gráfico_35"
   TextField "Campo de texto_9" at 123,12 size 125x25; Text 'Temperatura'
   TextField "Campo de texto_10" at 388,27 size 53x25; Text 'Flujo'
   TextField "Campo de texto_11" at 504,175 size 76x25; Text 'Presion'
   TextField "Campo de texto_12" at 560,10 size 201x25; Text 'Valvula Proporcional'
   TextField "Campo de texto_13" at 366,449 size 159x25; Text 'Velocidad Motor'
   TextField "Campo de texto_14" at 939,171 size 53x25; Text 'Nivel'
   IOField "Campo ES_4" at 248,12 size 96x32; FormatPattern s999999999.999
      ProcessValue <- "temperatura"
   IOField "Campo ES_5" at 366,57 size 96x32; FormatPattern s999999999.999
      ProcessValue <- "flujo"
   IOField "Campo ES_6" at 608,40 size 96x32; FormatPattern s99999
      ProcessValue <- "valvula"
   IOField "Campo ES_7" at 395,476 size 96x32; FormatPattern s99999
      ProcessValue <- "bomba"
   Circle "Círculo_5" at 188,194 size 28x28
      Appearance <- "on_temp"
   IOField "Campo ES_8" at 500,147 size 96x32; FormatPattern s999999999.999
      ProcessValue <- "presion"
   Button "Botón_3" at 161,622 size 300x80; TextOff 'TENDENCIAS'
      on Click: ActivateScreen("tendencia on-off temperatura", 0)
   TextField "Campo de texto_3" at 88,434 size 102x32; Text 'ACTUAL'
   TextField "Campo de texto_4" at 69,68 size 133x32; Text 'CONTROL'
   TextField "Campo de texto_5" at 40,98 size 191x32; Text 'TEMPERATURA'
   TextField "Campo de texto_6" at 85,128 size 101x32; Text 'ON-OFF'
   Button "Botón_5" at 1024,75 size 61x79; TextOff 'Text'
      on Click: InvertBit("v3 llen")
   Button "Botón_6" at 1101,243 size 61x79; TextOff 'Text'
      on Click: InvertBit("v3")
   Button "Botón_7" at 681,251 size 61x79; TextOff 'Text'
      on Click: InvertBit("v1llen")
   Button "Botón_8" at 790,252 size 61x79; TextOff 'Text'
      on Click: InvertBit("v2llen")
   Button "Botón_9" at 803,433 size 61x79; TextOff 'Text'
      on Click: InvertBit("v2vac")
   Button "Botón_10" at 693,432 size 61x79; TextOff 'Text'
      on Click: InvertBit("v1vac")
   Button "Botón_11" at 282,365 size 80x80; TextOff 'Text'
      on Click: InvertBit("calefactora")
   Button "Botón_12" at 280,218 size 80x80; TextOff 'Text'
      on Click: InvertBit("enfriadora")
   Circle "Círculo_1" at 712,405 size 23x23
      Appearance <- "Abrir Valvula Vaciado Tanque 1"
   Circle "Círculo_2" at 821,405 size 23x23
      Appearance <- "Abrir Valvula Vaciado Tanque 2"
   Circle "Círculo_3" at 700,227 size 23x23
      Appearance <- "Abrir Valvula Llenado Tanque 1"
   Circle "Círculo_4" at 809,225 size 23x23
      Appearance <- "Abrir Valvula Llenado Tanque 2"
   Button "Botón_4" at 1124,490 size 104x70; TextOff 'MANUAL'
      on Click: InvertBit("onproc")
   Button "Botón_14" at 383,511 size 120x84; TextOff 'Text'
      on Click: InvertBit("d7")

screen "parametros fuzzy flujo" 1280x740
   Button "Botón_1" at 1064,632 size 204x90; TextOff 'REGRESAR'
      on Click: ActivateScreen("fuzzy flujo", 0)
   TextField "Campo de texto_1" at 511,104 size 253x25; Text 'UNIVERSOS DE DISCURSO'
   TextField "Campo de texto_2" at 346,157 size 69x25; Text 'ERROR'
   TextField "Campo de texto_3" at 785,157 size 216x25; Text 'DERIVADA DEL ERROR'
   TextField "Campo de texto_4" at 167,211 size 109x25; Text 'NEGATIVO'
   TextField "Campo de texto_5" at 208,262 size 55x25; Text 'CERO'
   TextField "Campo de texto_6" at 172,321 size 98x25; Text 'POSITIVO'
   TextField "Campo de texto_7" at 682,211 size 109x25; Text 'NEGATIVO'
   TextField "Campo de texto_8" at 723,262 size 55x25; Text 'CERO'
   TextField "Campo de texto_9" at 687,321 size 98x25; Text 'POSITIVO'
   IOField "Campo ES_1" at 272,203 size 80x40; FormatPattern s999999999.999
      ProcessValue <- "EN_1"
   IOField "Campo ES_2" at 360,203 size 80x40; FormatPattern s999999999.999
      ProcessValue <- "EN_2"
   IOField "Campo ES_3" at 448,203 size 80x40; FormatPattern s999999999.999
      ProcessValue <- "EN_3"
   IOField "Campo ES_4" at 537,203 size 80x40; FormatPattern s999999999.999
      ProcessValue <- "EN_4"
   IOField "Campo ES_5" at 272,255 size 80x40; FormatPattern s999999999.999
      ProcessValue <- "EZ_1"
   IOField "Campo ES_6" at 360,255 size 80x40; FormatPattern s999999999.999
      ProcessValue <- "EZ_2"
   IOField "Campo ES_7" at 448,255 size 80x40; FormatPattern s999999999.999
      ProcessValue <- "EZ_3"
   IOField "Campo ES_8" at 537,255 size 80x40; FormatPattern s999999999.999
      ProcessValue <- "EZ_4"
   IOField "Campo ES_9" at 272,314 size 80x40; FormatPattern s999999999.999
      ProcessValue <- "EP_1"
   IOField "Campo ES_10" at 360,314 size 80x40; FormatPattern s999999999.999
      ProcessValue <- "EP_2"
   IOField "Campo ES_11" at 448,314 size 80x40; FormatPattern s999999999.999
      ProcessValue <- "EP_3"
   IOField "Campo ES_12" at 537,314 size 80x40; FormatPattern s999999999.999
      ProcessValue <- "EP_4"
   IOField "Campo ES_13" at 793,203 size 80x40; FormatPattern s999999999.999
      ProcessValue <- "DEN_1"
   IOField "Campo ES_14" at 884,203 size 80x40; FormatPattern s999999999.999
      ProcessValue <- "DEN_2"
   IOField "Campo ES_15" at 971,203 size 80x40; FormatPattern s999999999.999
      ProcessValue <- "DEN_3"
   IOField "Campo ES_16" at 1055,203 size 80x40; FormatPattern s999999999.999
      ProcessValue <- "DEN_4"
   IOField "Campo ES_17" at 793,255 size 80x40; FormatPattern s999999999.999
      ProcessValue <- "DEZ_1"
   IOField "Campo ES_18" at 793,314 size 80x40; FormatPattern s999999999.999
      ProcessValue <- "DEP_1"
   IOField "Campo ES_19" at 884,255 size 80x40; FormatPattern s999999999.999
      ProcessValue <- "DEZ_2"
   IOField "Campo ES_20" at 884,314 size 80x40; FormatPattern s999999999.999
      ProcessValue <- "DEP_2"
   IOField "Campo ES_21" at 971,255 size 80x40; FormatPattern s999999999.999
      ProcessValue <- "DEZ_3"
   IOField "Campo ES_22" at 971,314 size 80x40; FormatPattern s999999999.999
      ProcessValue <- "DEP_3"
   IOField "Campo ES_23" at 1055,255 size 80x40; FormatPattern s999999999.999
      ProcessValue <- "DEZ_4"
   IOField "Campo ES_24" at 1055,314 size 80x40; FormatPattern s999999999.999
      ProcessValue <- "DEP_4"

screen "plantilla" 1280x740
   GraphicView "Visor de gráficos_7" at 499,243 size 138x216; Picture "Gráfico_11"
   GraphicView "Visor de gráficos_2" at 924,449 size 56x50; Picture "Gráfico_14"
   GraphicView "Visor de gráficos_3" at 554,448 size 53x52; Picture "Gráfico_15"
   GraphicView "Visor de gráficos_4" at 632,290 size 52x29; Picture "Gráfico_16"
   GraphicView "Visor de gráficos_9" at 381,509 size 123x85; Picture "Gráfico_19"
   GraphicView "Visor de gráficos_10" at 388,97 size 61x52; Picture "Gráfico_20"
   GraphicView "Visor de gráficos_11" at 525,67 size 33x57; Picture "Gráfico_21"
   GraphicView "Visor de gráficos_12" at 628,83 size 61x63; Picture "Gráfico_22"
   GraphicView "Visor de gráficos_15" at 681,256 size 62x64; Picture "Gráfico_23"
   GraphicView "Visor de gráficos_17" at 748,469 size 55x58; Picture "Gráfico_24"
   GraphicView "Visor de gráficos_18" at 739,263 size 53x56; Picture "Gráfico_25"
   GraphicView "Visor de gráficos_6" at 790,256 size 62x64; Picture "Gráfico_23"
   GraphicView "Visor de gráficos_19" at 850,290 size 52x29; Picture "Gráfico_16"
   GraphicView "Visor de gráficos_20" at 894,243 size 138x216; Picture "Gráfico_11"
   GraphicView "Visor de gráficos_21" at 603,471 size 92x29; Picture "Gráfico_16"
   GraphicView "Visor de gráficos_22" at 692,437 size 62x64; Picture "Gráfico_23"
   GraphicView "Visor de gráficos_24" at 801,437 size 62x64; Picture "Gráfico_23"
   GraphicView "Visor de gráficos_25" at 861,471 size 67x29; Picture "Gráfico_16"
   GraphicView "Visor de gráficos_1" at 734,515 size 56x50; Picture "Gráfico_14"
   GraphicView "Visor de gráficos_8" at 495,537 size 251x29; Picture "Gráfico_16"
   GraphicView "Visor de gráficos_13" at 306,490 size 54x52; Picture "Gráfico_15"
   GraphicView "Visor de gráficos_14" at 344,513 size 48x29; Picture "Gráfico_16"
   GraphicView "Visor de gráficos_16" at 353,115 size 38x29; Picture "Gráfico_16"
   GraphicView "Visor de gráficos_23" at 445,116 size 187x29; Picture "Gráfico_16"
   GraphicView "Visor de gráficos_26" at 435,221 size 46x68; Picture "Gráfico_26"
   GraphicView "Visor de gráficos_27" at 434,333 size 46x68; Picture "Gráfico_26"
   GraphicView "Visor de gráficos_28" at 462,279 size 45x10; Picture "Gráfico_16"
   GraphicView "Visor de gráficos_29" at 463,391 size 45x10; Picture "Gráfico_16"
   GraphicView "Visor de gráficos_30" at 304,155 size 31x344; Picture "Gráfico_17"
   GraphicView "Visor de gráficos_31" at 307,117 size 52x48; Picture "Gráfico_27"
   GraphicView "Visor de gráficos_32" at 683,116 size 60x29; Picture "Gráfico_16"
   GraphicView "Visor de gráficos_34" at 750,153 size 31x120; Picture "Gráfico_17"
   IOField "Campo ES_1" at 1104,459 size 96x32; FormatPattern s99999
      ProcessValue <- "bomba"
   Circle "Círculo_1" at 712,405 size 23x23
      Appearance <- "v1vac"
   Circle "Círculo_2" at 821,405 size 23x23
      Appearance <- "v2vac"
   Circle "Círculo_3" at 700,227 size 23x23
      Appearance <- "v1llen"
   Circle "Círculo_4" at 809,225 size 23x23
      Appearance <- "v2llen"
   Bar "Barra_1" at 900,275 size 131x145; MinimumValue 0; MaximumValue 27000
      ProcessValue <- "Nivel tanque"
   GraphicView "Visor de gráficos_35" at 930,200 size 75x76; Picture "Gráfico_28"
   Circle "Círculo_6" at 647,144 size 23x23
      Appearance <- "d7"
   GraphicView "Visor de gráficos_37" at 282,217 size 80x80; Picture "Gráfico_30"
   Circle "Círculo_7" at 374,241 size 23x23
      Appearance <- "Activar Unidad Enfriadora"
   Circle "Círculo_8" at 379,403 size 23x23
      Appearance <- "Activar Unidad Calefactora"
   GraphicView "Visor de gráficos_36" at 282,365 size 80x80; Picture "Gráfico_31"
   Rectangle "Rectángulo_2" at 444,225 size 33x20
      Appearance <- "Switch de Nivel Alto Tanque 1 (NC)"
   Rectangle "Rectángulo_4" at 444,337 size 33x20
      Appearance <- "Switch de Nivel Bajo Tanque 1 (NO)"
   GraphicView "Visor de gráficos_5" at 1131,97 size 126x149; Picture "Gráfico_32"
   GraphicView "Visor de gráficos_33" at 1077,115 size 61x29; Picture "Gráfico_16"
   GraphicView "Visor de gráficos_38" at 1157,259 size 56x50; Picture "Gráfico_14"
   GraphicView "Visor de gráficos_39" at 1026,282 size 78x29; Picture "Gráfico_16"
   GraphicView "Visor de gráficos_40" at 1023,82 size 62x64; Picture "Gráfico_23"
   GraphicView "Visor de gráficos_41" at 1099,248 size 62x64; Picture "Gráfico_23"
   GraphicView "Visor de gráficos_42" at 1182,239 size 31x34; Picture "Gráfico_17"
   Circle "Círculo_9" at 1037,43 size 23x23
      Appearance <- "Abrir Valvula Llenado Tanque 3"
   GraphicView "Visor de gráficos_43" at 784,115 size 247x29; Picture "Gráfico_16"
   Circle "Círculo_10" at 1120,323 size 23x23
      Appearance <- "Abrir Valvula Vaciado Tanque 3"
   GraphicView "Visor de gráficos_44" at 739,117 size 53x53; Picture "Gráfico_34"
   GraphicView "Visor de gráficos_45" at 275,51 size 53x149; Picture "Gráfico_35"
   TextField "Campo de texto_9" at 123,12 size 125x25; Text 'Temperatura'
   TextField "Campo de texto_10" at 388,27 size 53x25; Text 'Flujo'
   TextField "Campo de texto_11" at 504,175 size 76x25; Text 'Presion'
   TextField "Campo de texto_12" at 560,10 size 201x25; Text 'Valvula Proporcional'
   TextField "Campo de texto_13" at 366,449 size 159x25; Text 'Velocidad Motor'
   TextField "Campo de texto_14" at 939,171 size 53x25; Text 'Nivel'
   Button "Botón_12" at 1122,515 size 61x79; TextOff 'Text'
      on Click: InvertBit("Abrir Valvula Vaciado Tanque 3")

screen "Variables fisicas" 1280x740
   TextField "Campo de texto_1" at 467,52 size 347x43; Text 'VARIABLES FISICAS'
   Button "Botón_1" at 91,166 size 337x113; TextOff 'PESO'
      on Click: ActivateScreen("controles peso", 0)
   Button "Botón_2" at 471,166 size 337x113; TextOff 'FLUJO'
      on Click: ActivateScreen("controles flujo", 0)
   Button "Botón_3" at 854,166 size 337x113; TextOff 'PRESION'
      on Click: ActivateScreen("controles presion", 0)
   Button "Botón_4" at 247,339 size 337x113; TextOff 'NIVEL'
      on Click: ActivateScreen("controles nivel", 0)
   Button "Botón_5" at 687,340 size 337x113; TextOff 'TEMPERATURA'
      on Click: ActivateScreen("controles temperatura", 0)
   Button "Botón_6" at 472,572 size 337x113; TextOff 'REGRESAR'
      on Click: ActivateScreen("Imagen raíz", 0)

screen "controles peso" 1280x740
   TextField "Campo de texto_1" at 331,52 size 619x43; Text 'TECNICAS DE CONTROL PARA PESO'
   Button "Botón_7" at 488,576 size 304x104; TextOff 'REGRESAR'
      on Click: ActivateScreen("Variables fisicas", 0)
   Button "Botón_3" at 482,339 size 304x122; TextOff 'ON-OFF'
      on Click: ActivateScreen("on-off peso", 0)

screen "controles presion" 1280x740
   TextField "Campo de texto_1" at 298,52 size 685x43; Text 'TECNICAS DE CONTROL PARA PRESION'
   Button "Botón_7" at 488,576 size 304x104; TextOff 'REGRESAR'
      on Click: ActivateScreen("Variables fisicas", 0)
   Button "Botón_2" at 482,167 size 304x122; TextOff 'PID'
      on Click: ActivateScreen("lgr presion", 0)
   Button "Botón_1" at 111,168 size 304x122; TextOff 'SINTONIZACION'
      on Click: ActivateScreen("sintonizacion presion", 0)
   Button "Botón_6" at 856,341 size 304x122; TextOff 'FUZZY'
      on Click: ActivateScreen("fuzzy presion", 0)

screen "controles nivel" 1280x740
   TextField "Campo de texto_1" at 329,52 size 624x43; Text 'TECNICAS DE CONTROL PARA NIVEL'
   Button "Botón_7" at 488,576 size 304x104; TextOff 'REGRESAR'
      on Click: ActivateScreen("Variables fisicas", 0)
   Button "Botón_2" at 482,167 size 304x122; TextOff 'PID'
      on Click: ActivateScreen("lgr nivel", 0)
   Button "Botón_3" at 482,339 size 304x122; TextOff 'ON-OFF'
      on Click: ActivateScreen("on-off nivel", 0)

screen "controles temperatura" 1280x740
   TextField "Campo de texto_1" at 249,52 size 784x43; Text 'TECNICAS DE CONTROL PARA TEMPERATURA'
   Button "Botón_7" at 488,576 size 304x104; TextOff 'REGRESAR'
      on Click: ActivateScreen("Variables fisicas", 0)
   Button "Botón_3" at 482,339 size 304x122; TextOff 'ON-OFF'
      on Click: ActivateScreen("on-off temperatura", 0)

